// TwinCAT 3 PLC project actuator
// Title: ESO LDC Actuator Library
// Company: ESO
// Author: Dan Popovic
// ProjectVersion: 1.0.0.2
// Description: Local Device Control - LDC Actuator Library based on State Machine
// ProgramVersion: 3.1.0.8
// libraries:
//   Tc2_Standard, * (Beckhoff Automation GmbH)
//   Tc2_System, * (Beckhoff Automation GmbH)
//   Tc2_Utilities, * (Beckhoff Automation GmbH)
//   Tc3_EventLogger, * (Beckhoff Automation GmbH)
//   Tc3_Module, * (Beckhoff Automation GmbH)
//   VisuDialogs, * (System)
// project tree:
//   DUTs/Enumerated/ E_ACTUATOR_RPC_ERROR.TcDUT, E_ACTUATOR_COMMAND.TcDUT, E_ACTUATOR_EVENT.TcDUT, E_ACTUATOR_ERROR.TcDUT, E_ACTUATOR_STATUS.TcDUT, E_ACTUATOR_STATE.TcDUT, E_ACTUATOR_HW_STATUS.TcDUT, E_ACTUATOR_SUBSTATE.TcDUT
//   DUTs/Structures/ T_ACTUATOR_CFG.TcDUT, T_SIM_ACTUATOR_CFG.TcDUT, T_ACTUATOR_CTRL.TcDUT, T_ACTUATOR_INFO.TcDUT, T_ACTUATOR_STAT.TcDUT, T_SIM_ACTUATOR_STAT.TcDUT
//   / GlobalTextList.TcGTLO, PlcTask.TcTTO, Visualization Manager.TcVMO (not stored)
//   POUs/ FB_SIM_ACTUATOR.TcPOU, FB_ACTUATOR.TcPOU, MAIN.TcPOU
//   Version/ Global_Version.TcGVL
//   VISUs/ GUI_Actuator001.TcVIS, GUI_Actuator002.TcVIS, GUI_Actuator003.TcVIS, GUI_Actuator004.TcVIS
//   VISUs/Templates/ GUI_TEMPLATE_ACTUATOR.TcVIS
// real-time tasks:
//   TASK PlcTask: cycle T#1ms, priority 20, ADS port 350
// variable links:
//   actuator/actuator Instance <-> actuator/actuator Instance
//     PlcTask Inputs/MAIN.Actuator001.i_bOn <-> PlcTask Outputs/MAIN.SIM_Actuator001.q_bOn
//     PlcTask Inputs/MAIN.Actuator002.i_bOn <-> PlcTask Outputs/MAIN.SIM_Actuator002.q_bOn
//     PlcTask Inputs/MAIN.Actuator002.i_nCouplerState <-> PlcTask Outputs/MAIN.SIM_Actuator002.q_nCouplerState
//     PlcTask Inputs/MAIN.Actuator003.i_nCouplerState <-> PlcTask Outputs/MAIN.SIM_Actuator003.q_nCouplerState
//     PlcTask Inputs/MAIN.Actuator004.i_nCouplerState <-> PlcTask Outputs/MAIN.SIM_Actuator004.q_nCouplerState
//     PlcTask Inputs/MAIN.SIM_Actuator001.i_bSwitch <-> PlcTask Outputs/MAIN.Actuator001.q_bSwitch
//     PlcTask Inputs/MAIN.SIM_Actuator002.i_bSwitch <-> PlcTask Outputs/MAIN.Actuator002.q_bSwitch
//     PlcTask Inputs/MAIN.SIM_Actuator003.i_bSwitch <-> PlcTask Outputs/MAIN.Actuator003.q_bSwitch
//     PlcTask Outputs/MAIN.Actuator004.q_bSwitch <-> PlcTask Inputs/MAIN.SIM_Actuator004.i_bSwitch
//     PlcTask Outputs/MAIN.SIM_Actuator001.q_nCouplerState <-> PlcTask Inputs/MAIN.Actuator001.i_nCouplerState
//     PlcTask Outputs/MAIN.SIM_Actuator003.q_bOn <-> PlcTask Inputs/MAIN.Actuator003.i_bOn
//     PlcTask Outputs/MAIN.SIM_Actuator004.q_bOn <-> PlcTask Inputs/MAIN.Actuator004.i_bOn

CONFIGURATION actuator
    RESOURCE PLC ON TwinCAT3
        TASK PlcTask(INTERVAL := T#1ms, PRIORITY := 20);
        PROGRAM MAIN WITH PlcTask : MAIN;
    END_RESOURCE
END_CONFIGURATION

// ---- DUTs/Enumerated/E_ACTUATOR_RPC_ERROR.TcDUT
{attribute 'qualified_only'}
{attribute 'strict'}
TYPE E_ACTUATOR_RPC_ERROR :
(
	OK						:= 0,
	NOT_OP					:= -1,			
	NOT_NOTOP_READY			:= -2,			
	NOT_NOTOP				:= -3,			
	SWITCHING_ON			:= -4,			
	SWITCHING_OFF			:= -5,			
	LOCAL					:= -7			
);
END_TYPE

// ---- DUTs/Enumerated/E_ACTUATOR_COMMAND.TcDUT
{attribute 'qualified_only'}
{attribute 'strict'}
TYPE E_ACTUATOR_COMMAND :
(
	NONE	:= 0,
	
	RESET,
	INIT,
	STOP,
	ENABLE,
	DISABLE,
	ON,
	OFF
	
);
END_TYPE

// ---- DUTs/Enumerated/E_ACTUATOR_EVENT.TcDUT
{attribute 'qualified_only'}
{attribute 'strict'}
TYPE E_ACTUATOR_EVENT :
(
	NONE	:= 0,
	
	(* events corresponding to commands *)
	RESET,
	INIT,
	STOP,
	ENABLE,
	DISABLE,
	ON,
	OFF,
	
	(* 
		Events corresponding to internal events 
	*)
	
	INITON,		// Needed for detection of HW failures during initialisation
	INITOFF,
	DISABLEON,
	DISABLEOFF,
	
	(* events mapped to HW signals *)
	ISON,
	ISOFF,

	HWOK,
	ERRHW,
	ERRMAXON,
	ERRTIMEOUT,
	ERRINIT,
	ERRDISABLE
	
);
END_TYPE

// ---- DUTs/Enumerated/E_ACTUATOR_ERROR.TcDUT
{attribute 'qualified_only'}
{attribute 'strict'}
TYPE E_ACTUATOR_ERROR :
(
	OK					:= 0,
	HW_NOTOP,			
	WRONG_CMD,			
	INCONSISTENT,		
	INIT_FAILURE,		
	ENABLE_FAILURE,
	DISABLE_FAILURE,
	ON_FAILURE,
	OFF_FAILURE,
	FAILURE_SIG,
	MAXON,
	STILL_COOLING,
	TIMEOUT,
	// Simulator errors
	NOT_INITIALISED		:= 90,
	ZERO_POINTER		:= 100	
);
END_TYPE

// ---- DUTs/Enumerated/E_ACTUATOR_STATUS.TcDUT
{attribute 'qualified_only'}
{attribute 'strict'}
TYPE E_ACTUATOR_STATUS :
(
	OK	:= 0,
	ERROR
);
END_TYPE

// ---- DUTs/Enumerated/E_ACTUATOR_STATE.TcDUT
{attribute 'qualified_only'}
{attribute 'strict'}
TYPE E_ACTUATOR_STATE :
(
	NONE	:= 0,
	NOTOP,
	OP
);
END_TYPE

// ---- DUTs/Enumerated/E_ACTUATOR_HW_STATUS.TcDUT
{attribute 'qualified_only'}
{attribute 'strict'}
TYPE E_ACTUATOR_HW_STATUS :
(
	UNKNOWN	:= 0,
	ERROR,
	OFF,
	ON
);
END_TYPE

// ---- DUTs/Enumerated/E_ACTUATOR_SUBSTATE.TcDUT
{attribute 'qualified_only'}
{attribute 'strict'}
TYPE E_ACTUATOR_SUBSTATE :
(
	NONE					:= 0,
	
	NOTOP_NOTREADY			:= 100,
	NOTOP_READY_OFF			:= 103,
	NOTOP_READY_ON			:= 104,
	NOTOP_SWITCHING_OFF		:= 109,           
	NOTOP_SWITCHING_ON		:= 110,
	NOTOP_ERROR				:= 199,
	
	OP_OFF					:= 206,            
	OP_SWITCHING_OFF		:= 207,           
	OP_ON					:= 209,
	OP_SWITCHING_ON			:= 210,
	OP_ERROR				:= 299
);
END_TYPE

// ---- DUTs/Structures/T_ACTUATOR_CFG.TcDUT
TYPE T_ACTUATOR_CFG :
STRUCT
	sName:				STRING	:= 'Actuator';// Instance name
	bActiveLowOn:		BOOL 	:= FALSE;	(* If TRUE, On signal is Active Low *)
	bActiveLowSwitch:	BOOL 	:= FALSE;	(* If TRUE, Switch ctrl signal is Active Low *)

	bAutoOp:			BOOL 	:= FALSE;	// If TRUE, go automatically to OPERATIONAL state
	bInitialState:		BOOL 	:= FALSE;	(* default power state is OFF *)
	bInvertAnalog:		BOOL 	:= FALSE;	(* If TRUE, analog feedback is active, if signal < nAnalogThreshold *)
	
	nAnalogThreshold:	DINT 	:= 0;		(* Analog feedback signal threshold [bits].
										   If this signal is used, any value above it will indicate that the power is ON. *)

	nMaxOn:				UDINT 	:= 0;		(* Maximum time for power to be ON [sec] *)
	nSigStablePeriod:   UDINT 	:= 200;		(* signal is stable if it has been constant for so long [msec] *)
	nTimeout:     		UDINT 	:= 5000;	(* timeout for state transitions [msec] *)

	// Logging
	bLogExtTime:		BOOL 	:= FALSE;		// If TRUE, use external time in event logs. Default FALSE.
	bDebug:				BOOL 	:= FALSE;		// If TRUE, show event logs of Debug type. Default FALSE.
	bLog:				BOOL 	:= TRUE;		// If TRUE, log events. Default TRUE.


	
END_STRUCT
END_TYPE

// ---- DUTs/Structures/T_SIM_ACTUATOR_CFG.TcDUT
TYPE T_SIM_ACTUATOR_CFG :
STRUCT
	bActiveLowOn:		BOOL := FALSE;
	bActiveLowSwitch:	BOOL := FALSE;

	nDelay:     		UDINT := 1000;	(* Simulated delay for commands [msec] *)
	
END_STRUCT
END_TYPE

// ---- DUTs/Structures/T_ACTUATOR_CTRL.TcDUT
TYPE T_ACTUATOR_CTRL :
STRUCT
	nCommand:		DINT	:= E_ACTUATOR_COMMAND.NONE;	(* See E_ACTUATOR_COMMAND *)
	bExecute:		BOOL;
	
END_STRUCT
END_TYPE

// ---- DUTs/Structures/T_ACTUATOR_INFO.TcDUT
TYPE T_ACTUATOR_INFO :
STRUCT
(*
Driver Information 

Change Log:
*)
	sDate:			STRING(32)	:= '2018-10-26';
	sDescription:	STRING(80) 	:= 'State Machine based Actuator controller';
	sName:			STRING(64)	:= 'FB_ACTUATOR';
	sPlatform:		STRING(32)	:= 'CoDeSys';
	sSynopsis:		STRING(64)	:= 'State Machine based Actuator controller';
	nVersionMajor:	DINT		:= 1;
	nVersionMinor:	DINT		:= 0;
END_STRUCT
END_TYPE

// ---- DUTs/Structures/T_ACTUATOR_STAT.TcDUT
TYPE T_ACTUATOR_STAT :
STRUCT
	bLocal:			BOOL	:= FALSE;						(* if TRUE, device operated from PLC GUI *)

	nLastCommand:	DINT	:= E_ACTUATOR_COMMAND.NONE;			(* Last command sent to the device *)

	nErrorCode: 	DINT 	:= E_ACTUATOR_ERROR.HW_NOTOP;		(* Error code *)
	nHwStatus: 		DINT	:= E_ACTUATOR_HW_STATUS.UNKNOWN; 		(* Unknown, error, on, of. See E_ACTUATOR_HW_STATUS *)
	nRpcErrorCode: 	DINT	:= E_ACTUATOR_RPC_ERROR.OK;		(* RPC Error code *)
	nStatus: 		DINT	:= E_ACTUATOR_STATUS.ERROR; 			(* Device status *)

	sErrorText: 	STRING 	:= 'OK'; 						(* Error text *)
	sHwStatus: 		STRING 	:= 'UNKNOWN'; 					(* HW Status in textual form: 'UNKNOWN', 'ERROR', 'OPEN' or 'CLOSED' *)
	sLastCommand:	STRING	:= 'NONE';						(* Last command, as string, sent to the device *)
	sLibVersion:	STRING	:= 'UNKNOWN';					(* Library version as string, e.g. '1.2.0.0' *)
	sRPCErrorText: 	STRING 	:= 'OK'; 						(* RPC Error text *)
	sStatus: 		STRING 	:= 'OK'; 						(* Status in textual form, e.g. 'OFF' *)
	
	sState:			STRING	:= 'NOT OP';
	sSubstate:		STRING	:= 'NOT READY';
	
	nState:			E_ACTUATOR_STATE		:= E_ACTUATOR_STATE.NOTOP;
	nSubstate:		E_ACTUATOR_SUBSTATE	:= E_ACTUATOR_SUBSTATE.NOTOP_NOTREADY;
	
	sActionDesc:	STRING	:= '';
	sEventDesc:		STRING	:= '';

	


	nCycleCounter:		UDINT	:= 0;
	nCycleTime:			UDINT	:= 0;						// Cycle time in us (microsec)

	nTimeOn: 			UDINT 	:= 0;						(* Time power has been ON since last ON command [sec] *)
	nTimeOnStart:		UDINT 	:= 0;						(* Absolute start time of last power ON command [sec] *)
	nTimeOnTotal:		UDINT 	:= 0;						(* Total time power has been ON [sec] *)
	nTimeOnTotalStart:	UDINT 	:= 0;						(* Absolute start time of power ON [sec] *)
	nTimeOff: 			UDINT 	:= 0;						(* Time power has been OFF [sec] *)
	nTimeOffStart:		UDINT 	:= 0;						(* Time power has been OFF [sec] *)
	
END_STRUCT
END_TYPE

// ---- DUTs/Structures/T_SIM_ACTUATOR_STAT.TcDUT
TYPE T_SIM_ACTUATOR_STAT :
STRUCT
	bInitialised:	BOOL	:= FALSE;						(* If TRUE, power simulator is initialised *)

	nErrorCode: 	DINT 	:= E_ACTUATOR_ERROR.NOT_INITIALISED;	(* Error code *)
	sErrorText: 	STRING 	:= 'NOT INITIALISED'; 			(* Error text *)
	sStatus: 		STRING 	:= 'ERROR'; 					(* power status in textual form, e.g. 'OFF' *)
END_STRUCT
END_TYPE

// ---- Version/Global_Version.TcGVL
{attribute 'TcGenerated'}
{attribute 'no-analysis'}
{attribute 'linkalways'}
// This function has been automatically generated from the project information.
VAR_GLOBAL CONSTANT
	{attribute 'const_non_replaced'}
	stLibVersion_ESO_LDC_Actuator_Library : ST_LibVersion := (iMajor := 1, iMinor := 0, iBuild := 0, iRevision := 2, nFlags := 0, sVersion := '1.0.0.2');
END_VAR

// ---- POUs/MAIN.TcPOU
PROGRAM MAIN
VAR
	
	{attribute 'OPC.UA.DA':='1'}
	Actuator001:		FB_ACTUATOR;	// Simulated power always
	{attribute 'OPC.UA.DA':='1'}
	Actuator002:		FB_ACTUATOR;	// Simulated power always
	{attribute 'OPC.UA.DA':='1'}
	Actuator003:		FB_ACTUATOR;	// Real power if connected to a PLC
	{attribute 'OPC.UA.DA':='1'}
	Actuator004:		FB_ACTUATOR;	// Real power if connected to a PLC

	{attribute 'OPC.UA.DA':='1'}
	SIM_Actuator001:	FB_SIM_ACTUATOR;
	{attribute 'OPC.UA.DA':='1'}
	SIM_Actuator002:	FB_SIM_ACTUATOR;
	{attribute 'OPC.UA.DA':='1'}
	SIM_Actuator003:	FB_SIM_ACTUATOR;
	{attribute 'OPC.UA.DA':='1'}
	SIM_Actuator004:	FB_SIM_ACTUATOR;
	
END_VAR

// Actuator001 configuration:
// - Go to  OPERATIONAL on PLC reboot
// - Initial state is OFF
Actuator001(in_sName:='Actuator001', in_bAutoOp:=TRUE,in_bInitialState:=FALSE);

// Actuator002 configuration:
// - Go to  OPERATIONAL on PLC reboot
// - Initial state is ON
Actuator002(in_sName:='Actuator002', in_bAutoOp:=TRUE,in_bInitialState:=TRUE);

// Actuator003 configuration:
// - Remain in NOTOP on PLC reboot
// - Initial state is OFF
Actuator003(in_sName:='Actuator003', in_bAutoOp:=FALSE,in_bInitialState:=FALSE);

// Actuator004 configuration:
// - Go to  OPERATIONAL on PLC reboot
// - Initial state is ON
Actuator004(in_sName:='Actuator004', in_bAutoOp:=TRUE,in_bInitialState:=TRUE);


// Actuator001 Simulator
SIM_Actuator001(ptrDev:=ADR(Actuator001));
// Actuator002 Simulator
SIM_Actuator002(ptrDev:=ADR(Actuator002));
// Actuator003 Simulator
SIM_Actuator003(ptrDev:=ADR(Actuator003));
// Actuator004 Simulator
SIM_Actuator004(ptrDev:=ADR(Actuator004));

END_PROGRAM

// ---- POUs/FB_ACTUATOR.TcPOU
FUNCTION_BLOCK FB_ACTUATOR
VAR_INPUT
	{attribute 'OPC.UA.DA' := '0'}
	in_sName:				STRING	:= 'Actuator';	// Default device name

	{attribute 'OPC.UA.DA' := '0'}
	in_bActiveLowOn:		BOOL	:= FALSE;	// If TRUE, On signal is Active Low. Default FALSE.
	{attribute 'OPC.UA.DA' := '0'}
	in_bActiveLowSwitch:	BOOL 	:= FALSE;	// If TRUE, Switch ctrl signal is Active Low. Default FALSE.

	{attribute 'OPC.UA.DA' := '0'}
	in_bAutoOp:				BOOL 	:= FALSE;	// If TRUE, go automatically to OPERATIONAL state. Default FALSE.
	{attribute 'OPC.UA.DA' := '0'}
	in_bInitialState:		BOOL 	:= FALSE;	// Default power state is OFF (FALSE).
	{attribute 'OPC.UA.DA' := '0'}
	in_bInvertAnalog:		BOOL 	:= FALSE;	// If TRUE, analog feedback is active if signal < nAnalogThreshold. Default FALSE.
	
	{attribute 'OPC.UA.DA' := '0'}
	in_nAnalogThreshold:	DINT 	:= 0;		// Analog feedback signal threshold [bits]. Used if <>0. Default 0, i.e. not used.
												// If this signal is used, any value above it will indicate that the power is ON.
	{attribute 'OPC.UA.DA' := '0'}
	in_nMaxOn:				UDINT 	:= 0;		// Maximum time for power to be ON [sec]. Default 0, no limit.
	{attribute 'OPC.UA.DA' := '0'}
	in_nSigStablePeriod:	UDINT 	:= 200;		// Signal is stable if it has been constant for so long [msec]. Default 200 ms.
	{attribute 'OPC.UA.DA' := '0'}
	in_nTimeout:     		UDINT 	:= 5000;	// Timeout for state transitions [msec]. Default 5000 ms (5 sec).
END_VAR
VAR_OUTPUT
END_VAR
VAR
	{attribute 'OPC.UA.DA' := '1'}
	cfg:		T_ACTUATOR_CFG;	
	{attribute 'OPC.UA.DA' := '1'}
	ctrl:		T_ACTUATOR_CTRL;	
	{attribute 'OPC.UA.DA' := '1'}
	{attribute 'OPC.UA.DA.Access' := '1'}
	info:		T_ACTUATOR_INFO;				// ReadOnly
	{attribute 'OPC.UA.DA' := '1'}
	{attribute 'OPC.UA.DA.Access' := '1'}
	stat:		T_ACTUATOR_STAT;				// ReadOnly

	{attribute 'OPC.UA.DA' := '0'}
	nEvent:		      	DINT := E_ACTUATOR_EVENT.NONE;
	{attribute 'OPC.UA.DA' := '0'}
	nInternalEvent:		DINT := E_ACTUATOR_EVENT.NONE;
	
	// Operational Events
	{attribute 'OPC.UA.DA' := '0'}
	fbEventStart:	FB_TcMessage;
	{attribute 'OPC.UA.DA' := '0'}
	fbEventEnd:		FB_TcMessage;
	{attribute 'OPC.UA.DA' := '0'}
	fbEventError:	FB_TcMessage;
	{attribute 'OPC.UA.DA' := '0'}
	fbEventDebug:	FB_TcMessage;
	{attribute 'OPC.UA.DA' := '0'}
	fbEventGeneral:	FB_TcMessage;
	
	
	(***** Local variables *****)
	{attribute 'OPC.UA.DA' := '0'}
	bOn:		BOOL;						// Feedback - combination of digital and analog
	{attribute 'OPC.UA.DA' := '0'}
	toutCmd:	TON;
	{attribute 'OPC.UA.DA' := '0'}
	trg:		R_TRIG;
	{attribute 'OPC.UA.DA' := '0'}
	timer:		TON;						// Timer for measuring duration of events
	


	///// Physical signals - to be mapped!!! /////

	// Outputs
	{attribute 'OPC.UA.DA' := '0'}
	q_bSwitch 		AT %Q*: 		BOOL;	// power control digital output

	// Inputs	
	{attribute 'OPC.UA.DA' := '0'}
	i_nCouplerState	AT %I*: 		UINT;	// Link it to Coupler->InfoData->State
	{attribute 'OPC.UA.DA' := '0'}
	i_bOn 			AT %I*: 		BOOL;	// Digital feedback signal
	{attribute 'OPC.UA.DA' := '0'}
	i_nOn			AT %I*: 		INT;	// Analog feedback signal

	// Flag if the device is ready to receive commands.
	// It takes about 3.5 sec for the system to go OPERATIONAL.
	{attribute 'OPC.UA.DA' := '0'}
	bDeviceReady:		BOOL 	:= FALSE;
END_VAR

IF NOT bDeviceReady THEN
	// Set device Configuration
	M_Configure();
	RETURN;
END_IF

// Increment counter.
// This will be seen as 'alive' flag.
stat.nCycleCounter	:= stat.nCycleCounter + 1;



(* === Check for commands and internal events to be processed === *)
CheckForEvents();

(* === Process events according to the State Machine === *)
ProcessEvents();

METHOD ActionErrExecute
VAR
END_VAR
SetAction('ActionErrExecute');

IF nEvent = E_ACTUATOR_EVENT.ERRTIMEOUT THEN
	stat.nErrorCode		:= E_ACTUATOR_ERROR.ON_FAILURE;
	stat.sErrorText		:= 'ERROR: Timeout';	
END_IF
END_METHOD

METHOD ActionInitAbort
VAR_INPUT
END_VAR
SetAction('ActionInitAbort');

(* reply Error *)
stat.nErrorCode		:= E_ACTUATOR_ERROR.INIT_FAILURE;
stat.sErrorText		:= 'ERROR: INIT command aborted due to STOP or RESET.';

(* Reset the timer for the command *)
toutCmd(IN:=FALSE);
END_METHOD

METHOD ActionInitExecute
VAR_INPUT
END_VAR
VAR
	nCurrentTime:	UDINT;
END_VAR
SetAction('ActionInitExecute');

// Log event
M_LogEventStart('INIT');

(* reply OK *)
stat.nErrorCode		:= E_ACTUATOR_ERROR.OK;
stat.sErrorText		:= 'OK';

(* Reset the timer action *)
toutCmd(IN:=FALSE);

nCurrentTime			:= GetTimeInSec();
stat.nTimeOffStart		:= nCurrentTime;
UpdateTimes(bOnState:=FALSE, bRestart:=FALSE, bReset:=FALSE);

// Do not touch the outputs.
// Just change the state depending on the status
IF bOn THEN
	SetState(E_ACTUATOR_STATE.NOTOP, E_ACTUATOR_SUBSTATE.NOTOP_READY_ON);
ELSE
	SetState(E_ACTUATOR_STATE.NOTOP, E_ACTUATOR_SUBSTATE.NOTOP_READY_OFF);
END_IF
END_METHOD

METHOD ActionInitReject
VAR_INPUT
END_VAR
SetAction('ActionInitReject');

(* Reject an INIT command since another one is in progress. *)
(* do not reset the timer ... *)
END_METHOD

METHOD ActionMaxOnFailure
VAR_INPUT
END_VAR
(* code to initiate the switching OFF of the power *)
SetAction('ActionMaxOnFailure');

// Log event
M_LogEventError('Actuator maximum ON time exceeded.. Switched to OFF.');

(* Set the error *)
SetStatus(E_ACTUATOR_ERROR.MAXON,'ERROR: Actuator maximum ON time exceeded.');

UpdateTimes(bOnState:=FALSE, bRestart:=TRUE, bReset:=FALSE);


(* Switch power OFF *)
q_bSwitch	:= GetLogicalState(FALSE, cfg.bActiveLowSwitch);

(* 
	Reset signal trigger and its timer. 
	Next transition activity, e.g. ActivitySwitchingOff, will complete when the signal has been OFF 
	for longer than cfg.nSigStablePeriod [ms].
*)
trg(CLK:=FALSE);
timer(IN:=FALSE);	// Timer for stable signal lasting cfg.nSigStablePeriod

(* Restart the command timer *)
toutCmd(IN:=FALSE);
toutCmd(IN:=TRUE,PT:=UDINT_TO_TIME(cfg.nTimeout));
END_METHOD

METHOD ActionOffExecute
VAR_INPUT
END_VAR
(* code to initiate the switching OFF of the power *)
SetAction('ActionOffExecute');

// Log event
M_LogEventStart('OFF');

(* Clear the error *)
SetStatus(E_ACTUATOR_ERROR.OK,'OK');

UpdateTimes(bOnState:=FALSE, bRestart:=TRUE, bReset:=FALSE);


(* Actuator power OFF *)
q_bSwitch	:= GetLogicalState(FALSE, cfg.bActiveLowSwitch);

(* 
	Reset signal trigger and its timer. 
	Next transition activity, e.g. ActivitySwitchingOff, will complete when the signal has been OFF 
	for longer than cfg.nSigStablePeriod [ms].
*)
trg(CLK:=FALSE);
timer(IN:=FALSE);	// Timer for stable signal lasting cfg.nSigStablePeriod

(* Restart the command timer *)
toutCmd(IN:=FALSE);
toutCmd(IN:=TRUE,PT:=UDINT_TO_TIME(cfg.nTimeout));
END_METHOD

METHOD ActionOnExecute
VAR_INPUT
END_VAR
(* Code to initiate turning the power ON *)

SetAction('ActionOnExecute');

// Log event
M_LogEventStart('ON');

(* Clear the error *)
SetStatus(E_ACTUATOR_ERROR.OK,'OK');

(* Turn the control signal ON  *)
q_bSwitch	:= GetLogicalState(TRUE, cfg.bActiveLowSwitch);


(* 
	Reset signal trigger and its timer. 
	Next transition activity, e.g. ActivitySwitchingOn, will complete when the signal has been ON 
	for longer than cfg.nSigStablePeriod [ms].
*)
trg(CLK:=FALSE);
timer(IN:=FALSE);	// Timer for stable signal lasting cfg.nSigStablePeriod

(* Start the timer for command timeout of cfg.nTimeout *)
toutCmd(IN:=FALSE);	
toutCmd(IN:=TRUE,PT:=UDINT_TO_TIME(cfg.nTimeout));
END_METHOD

METHOD ActionResetExecute
VAR_INPUT
END_VAR
SetAction('ActionResetExecute');

// Log event
M_LogEventStart('RESET');

(* reply Error *)
SetStatus(nErrorCode:=E_ACTUATOR_ERROR.OK, sErrorText:='OK');

// Go to the default state on PLC re-boot
q_bSwitch	:= GetLogicalState(cfg.bInitialState, cfg.bActiveLowSwitch);

// Reset ON/OFF times
UpdateTimes(bOnState:=bOn,bRestart:=FALSE,bReset:=TRUE);	

(* Reset the timer for the command *)
toutCmd(IN:=FALSE);

// In ActionOnExecute() and ActionOffExecute(), we are waiting for trg() to go from FALSE to TRUE.
// Trigger it with FALSE.
trg(CLK:=FALSE);

IF cfg.bInitialState = TRUE THEN
	ActionOnExecute();
	SetState(E_ACTUATOR_STATE.NOTOP, E_ACTUATOR_SUBSTATE.NOTOP_SWITCHING_ON);
ELSE
	ActionOffExecute();
	SetState(E_ACTUATOR_STATE.NOTOP, E_ACTUATOR_SUBSTATE.NOTOP_SWITCHING_OFF);
END_IF
END_METHOD

METHOD ActionUnexpExecute
VAR
END_VAR
SetAction('ActionUnexpExecute');

IF nEvent = E_ACTUATOR_EVENT.ISON THEN
	IF	stat.nLastCommand = E_ACTUATOR_COMMAND.ON 	AND
		stat.nSubstate = E_ACTUATOR_SUBSTATE.OP_OFF 	AND
		stat.nErrorCode = E_ACTUATOR_ERROR.TIMEOUT		THEN
		M_LogEventGeneral('Recovered after timeout. Actuator is ON');
	END_IF
ELSIF nEvent = E_ACTUATOR_EVENT.ISOFF THEN
	IF	stat.nLastCommand = E_ACTUATOR_COMMAND.OFF 	AND
		stat.nSubstate = E_ACTUATOR_SUBSTATE.OP_ON 	AND
		stat.nErrorCode = E_ACTUATOR_ERROR.TIMEOUT		THEN
		M_LogEventGeneral('Recovered after timeout. Actuator is OFF');
	END_IF
ELSIF nEvent = E_ACTUATOR_EVENT.ON THEN
	stat.nErrorCode		:= E_ACTUATOR_ERROR.STILL_COOLING;
	stat.sErrorText		:= 'ERROR: ON command not allowed while cooling.';	
	stat.sStatus		:= 'ERROR';	
	stat.nStatus		:= E_ACTUATOR_STATUS.ERROR;
END_IF
END_METHOD

METHOD ActivityOff
VAR_INPUT
END_VAR
SetAction('ActivityOff');

// Update the OFF time
UpdateTimes(bOnState:=FALSE, bRestart:=FALSE, bReset:=FALSE);
END_METHOD

METHOD ActivityOn
VAR_INPUT
END_VAR
SetAction('ActivityOn');

// Update the ON time
UpdateTimes(bOnState:=TRUE, bRestart:=FALSE, bReset:=FALSE);
END_METHOD

METHOD ActivitySwitchingOff
VAR_INPUT
END_VAR
(* 
	This activity monitors the OFF power task and 
	triggers the ISOFF event at completion. 
*)
SetAction('ActivitySwitchingOff');


(* 
	The signal has to be OFF for longer than cfg.nSigStablePeriod [msec].
	The timer will start when bOn=FALSE trigger is detected.
*)
(* Execute trigger - note the 'NOT bOn' detectiong the transition from ON to OFF *)
trg(CLK := NOT bOn);

IF trg.Q THEN
	(* Restart the signal duration timer *)
	timer(IN:=FALSE);
	timer(IN:=TRUE,PT:=UDINT_TO_TIME(cfg.nSigStablePeriod));
END_IF

(* Execute signal duration timer *)
timer();

IF	timer.Q OR 
	((NOT bOn) AND cfg.nSigStablePeriod = 0) THEN
	timer(IN:=FALSE);	// Reset the signal duration timer
	toutCmd(IN:=FALSE);	// Reset the command timeout timer

	(* Update time ON/OFF *)
	UpdateTimes(bOnState:=TRUE, bRestart:=FALSE, bReset:=FALSE);

	(* 
		Normally, we would go to state E_SWITCH_SUBSTATE.OP_COOLING. 
		However, if the cooldown time is zero, i.e. no cooldown, we go directly to state E_ACTUATOR_SUBSTATE.OP_OFF.
	*)
	nInternalEvent 		:= E_ACTUATOR_EVENT.ISOFF;
	
	// Log event
	M_LogEventEnd('OFF');

//	stat.nErrorCode		:= E_ACTUATOR_ERROR.OK;
//	stat.sErrorText		:= 'OK';	

	RETURN;
END_IF

(* 
	if the timeout is detected before reaching the position, 
	then trigger the internal error event 
*)
toutCmd();
IF toutCmd.Q THEN
	toutCmd(IN:=FALSE);	(* Reset Timer *)
	timer(IN:=FALSE);	(* Reset the signal duration timer *)
	
	nInternalEvent  := E_ACTUATOR_EVENT.ERRTIMEOUT;
	SetStatus(E_ACTUATOR_ERROR.TIMEOUT, 'ERROR: Switching OFF timed out.');

	// Log event
	M_LogEventError('OFF command timed out');
END_IF
END_METHOD

METHOD ActivitySwitchingOn
VAR_INPUT
END_VAR
(* 
	This activity to monitor the ON power task and 
	trigger the ISON event at completion. 
*)
SetAction('ActivitySwitchingOn');

(* 
	The signal has to be ON for longer than cfg.nSigStablePeriod [msec].
	The timer will start when bOn trigger is detected.
*)
(* Execute trigger *)
trg(CLK:=bOn);

IF trg.Q THEN
	(* Restart the signal duration timer *)
	timer(IN:=FALSE);
	timer(IN:=TRUE,PT:=UDINT_TO_TIME(cfg.nSigStablePeriod));
END_IF

(* Execute signal duration timer *)
timer();

IF	timer.Q OR 
	(bOn AND cfg.nSigStablePeriod = 0) THEN
	timer(IN:=FALSE);	// Reset the signal duration timer
	toutCmd(IN:=FALSE);	// Reset the command timeout timer

	(* Update time ON/OFF *)
	IF stat.nTimeOn > 0 THEN
		// power was already ON, restart the ON time.
		UpdateTimes(bOnState:=TRUE, bRestart:=TRUE, bReset:=FALSE);
	ELSE
		// power was OFF, don't restart the ON time.
		UpdateTimes(bOnState:=TRUE, bRestart:=FALSE, bReset:=FALSE);
	END_IF

	(* 
		Normally, we would go to state E_ACTUATOR_SUBSTATE.OP_WARMING. 
		However, if the warmup time is zero, i.e. no warmup, we go directly to state E_ACTUATOR_SUBSTATE.OP_ON.
	*)
	nInternalEvent 		:= E_ACTUATOR_EVENT.ISON;	
	
	// Log event
	M_LogEventEnd('ON');

	stat.nErrorCode		:= E_ACTUATOR_ERROR.OK;
	stat.sErrorText		:= 'OK';	

	RETURN;
END_IF

(* 
	if the timeout is detected before reaching the position, 
	then trigger the internal error event 
*)
toutCmd();
IF toutCmd.Q THEN
	toutCmd(IN:=FALSE);	(* Reset Timer *)
	timer(IN:=FALSE);	(* Reset the signal duration timer *)
	
	nInternalEvent  := E_ACTUATOR_EVENT.ERRTIMEOUT;
	SetStatus(E_ACTUATOR_ERROR.TIMEOUT, 'ERROR: Switching ON timed out.');

	// Log event
	M_LogEventError('ON command timed out');

END_IF
END_METHOD

METHOD CheckForEvents
VAR_INPUT
END_VAR

(* 
	Start assuming the HW is OK. 
	This is needed to recover from the situation where 
	the HW was failing and now it is working.
*)
nEvent := E_ACTUATOR_EVENT.HWOK;


(*
	Read all inputs, i.e. get status of INPUT signals based on ActiveLow configuration 
*)


(* The power ON feedback can be analog and/or digital. *)
IF 	(GetLogicalState(i_bOn, cfg.bActiveLowOn)) OR
	(cfg.nAnalogThreshold <> 0 AND (i_nOn > cfg.nAnalogThreshold) AND NOT cfg.bInvertAnalog) OR
	(cfg.nAnalogThreshold <> 0 AND (i_nOn < cfg.nAnalogThreshold) AND     cfg.bInvertAnalog)	THEN
	bOn	:= TRUE;
ELSE
	bOn	:= FALSE;
END_IF


UpdateTimes(bOnState:=bOn,bRestart:=FALSE, bReset:=FALSE);	// Update the Time


(* HW Status in textual form: 'ERROR', 'ON' or 'OFF' *)
IF 		bOn   = TRUE  THEN
	stat.nHwStatus	:= E_ACTUATOR_HW_STATUS.ON;
	stat.sHwStatus	:= 'ON';
ELSIF 	bOn   = FALSE  THEN
	stat.nHwStatus	:= E_ACTUATOR_HW_STATUS.OFF;
	stat.sHwStatus	:= 'OFF';
END_IF

(* 
	Check for events in the following order: 
   	1) HW failure: without HW avilability there is no point to do anything
	2) Internal events: to allow completing the initiated commands before 
                        starting processing new commands. 
   	3) Commands: to react to external commands. Commands should be executed 
                 before processing HW signals to allow to start a recovery action.
   	4) HW signals:  such as power is ON/OFF.
*)

IF i_nCouplerState <> 8 THEN	
	(* Check if the HW is NOT OK *)
	(*
	If the hardware status is NOT OK, we cannot trust the readings.
	Variable i_nCouplerState has to be mapped to a State of a terminal, e.g. EK1100.
	The value should be 8.
 	*)
	SetEvent(E_ACTUATOR_EVENT.ERRHW);
	SetStatus(E_ACTUATOR_ERROR.HW_NOTOP, 'ERROR: HW not in OPERATIONAL state');
	RETURN;

ELSIF nInternalEvent <> E_ACTUATOR_EVENT.NONE THEN
	(* Handle internal events *)
	SetEvent(nInternalEvent);
	nInternalEvent := E_ACTUATOR_EVENT.NONE;
ELSIF ctrl.bExecute = TRUE  THEN
	(* Handle commands *)
	ctrl.bExecute		:= FALSE;			(* Clear the Execute bit *)
	SetLastCommand(ctrl.nCommand);			(* Save the last command *)
	SetEvent(ctrl.nCommand);
	ctrl.nCommand 		:= E_ACTUATOR_COMMAND.NONE;	(* Clear the Command *)
ELSE
	(* Handle HW problems and unexpected bahaviour *)
	
	IF stat.nSubstate = E_ACTUATOR_SUBSTATE.NOTOP_READY_OFF OR 
	   stat.nSubstate = E_ACTUATOR_SUBSTATE.NOTOP_READY_ON OR 
	   stat.nSubstate = E_ACTUATOR_SUBSTATE.OP_OFF OR 
	   stat.nSubstate = E_ACTUATOR_SUBSTATE.OP_ON OR 
	   stat.nSubstate = E_ACTUATOR_SUBSTATE.OP_ERROR THEN
	   
		(* Set events for ON and OFF *)		
		IF	bOn   = TRUE  THEN
			SetEvent(E_ACTUATOR_EVENT.ISON);
		ELSIF	bOn   = FALSE THEN
			SetEvent(E_ACTUATOR_EVENT.ISOFF);
		END_IF	
	END_IF	
(*
	IF stat.nSubstate = E_ACTUATOR_SUBSTATE.OP_SWITCHING_ON THEN
		(* Set events for ON  *)		
		IF	bOn   = TRUE  THEN
			SetEvent(E_ACTUATOR_EVENT.ISON);
		END_IF	
	END_IF	
	*)
END_IF
END_METHOD

METHOD GetLogicalState : BOOL
(*
	This method returns the state of the variable based on its 
	activeLow configuration.
	Syntax:
		bState	:= GetLogicalState (<var value>,  <activeLow cfg>);
		
	Example 1:
		var = TRUE;
		activeLow = FALSE;
		bState	:= GetLogicalState (TRUE,  FALSE); = TRUE

	Example 2:
		var = TRUE;
		activeLow = TRUE;
		bState	:= GetLogicalState (TRUE,  TRUE); = FALSE
*)
VAR_INPUT
	state:		BOOL;
	activeLow:	BOOL;
END_VAR
IF activeLow THEN
	GetLogicalState := NOT state;
ELSE
	GetLogicalState := state;
END_IF
END_METHOD

METHOD GetTimeInSec : UDINT
(*
	This method returns absolute time in seconds.
*)
(* System time is given in 100ns. Divide by 10000000 to get in seconds. *)
GetTimeInSec := ULINT_TO_UDINT(Tc2_System.F_GetSystemTime() / 10000000);
END_METHOD

METHOD M_Configure : BOOL
VAR_INPUT
END_VAR
VAR
     fbGetCurTaskIdx:	GETCURTASKINDEX;
END_VAR
// If device is ready, there is nothing to configure.
IF bDeviceReady THEN
	RETURN;
END_IF

// If first cycle, copy configuration AND RETURN in order for the system to read all inputs before doing any work
IF stat.nCycleCounter = 0 THEN
	
	// Copy input parameters into configuration
	cfg.sName				:=	in_sName;			

	cfg.bActiveLowOn		:= in_bActiveLowOn;
	cfg.bActiveLowSwitch	:= in_bActiveLowSwitch;
	cfg.bAutoOp				:= in_bAutoOp;
	cfg.bInitialState		:= in_bInitialState;
	cfg.bInvertAnalog		:= in_bInvertAnalog;
	cfg.nAnalogThreshold	:= in_nAnalogThreshold;
	cfg.nMaxOn				:= in_nMaxOn;
	cfg.nSigStablePeriod	:= in_nSigStablePeriod;
	cfg.nTimeout			:= in_nTimeout;
	
	// Get the version number 
	stat.sLibVersion	:= stLibVersion_ESO_LDC_Actuator_Library.sVersion;

	// Get cycle time in microsec.
	// CycleTime in _TaskInfo is given in 100 ns. 1 us = 1000 ns
	fbGetCurTaskIdx();
	stat.nCycleTime	:=  (TwinCAT_SystemInfoVarList._TaskInfo[fbGetCurTaskIdx.index].CycleTime)/10;
	
	// Increment counter.
	stat.nCycleCounter	:= stat.nCycleCounter + 1;
	RETURN;
ELSIF (stat.nCycleCounter * stat.nCycleTime) < 5000000 THEN
	// EtherCAT is normally ready after 3.5 sec.
	// We give it 5 sec to consider it to be ready.
	// Increment counter.
	stat.nCycleCounter	:= stat.nCycleCounter + 1;
	RETURN;
END_IF


// Create Event instances
fbEventStart.CreateEx	(TC_EVENTS.ActuatorOpsEventClass.ActionStart,0);
fbEventEnd.CreateEx		(TC_EVENTS.ActuatorOpsEventClass.ActionEnd,0);
fbEventError.CreateEx	(TC_EVENTS.ActuatorOpsEventClass.Error,0);
fbEventDebug.CreateEx	(TC_EVENTS.ActuatorOpsEventClass.Debug,0);
fbEventGeneral.CreateEx	(TC_EVENTS.ActuatorOpsEventClass.General,0);

// The device is ready now.
bDeviceReady := TRUE;


// Clear errors
stat.nErrorCode		:= E_ACTUATOR_ERROR.OK;
stat.sErrorText		:= 'OK';	


//
// Set next state based on cfg.bAutoOp
//

// Go to the default state on PLC re-boot.
// Default state is set in cfg.bInitialState.
q_bSwitch	:= GetLogicalState(cfg.bInitialState, cfg.bActiveLowSwitch);

// In ActionOnExecute() and ActionOffExecute(), we are waiting for trg() to go from FALSE to TRUE.
// Trigger it with FALSE.
trg(CLK:=FALSE);

// Go directly to the target state.
IF NOT cfg.bAutoOp THEN
	// Go automatically to NOTOP ON or OFF
	IF cfg.bInitialState = TRUE THEN
		ActionOnExecute();
		SetState(E_ACTUATOR_STATE.NOTOP, E_ACTUATOR_SUBSTATE.NOTOP_SWITCHING_ON);
	ELSE
		ActionOffExecute();
		SetState(E_ACTUATOR_STATE.NOTOP, E_ACTUATOR_SUBSTATE.NOTOP_SWITCHING_OFF);
	END_IF
ELSE
	// Go automatically to OPERATIONAL
	// If initial state is ON, go to E_ACTUATOR_SUBSTATE.OP_SWITCHING_ON.
	// Otherwise, go to E_ACTUATOR_SUBSTATE.OP_SWITCHING_OFF.
	IF cfg.bInitialState = TRUE THEN
		ActionOnExecute();
		SetState(E_ACTUATOR_STATE.OP, E_ACTUATOR_SUBSTATE.OP_SWITCHING_ON);
	ELSE
		ActionOffExecute();
		SetState(E_ACTUATOR_STATE.OP, E_ACTUATOR_SUBSTATE.OP_SWITCHING_OFF);
	END_IF
END_IF
END_METHOD

METHOD M_GetRpcErrorText : STRING
VAR_INPUT
	ErrorCode:	INT;
END_VAR
VAR
	str:	STRING;
END_VAR
CASE ErrorCode OF
	E_ACTUATOR_RPC_ERROR.OK:					str	:= 'OK';
	E_ACTUATOR_RPC_ERROR.NOT_OP:				str	:= 'Cannot control device. Not in OP state.';
	E_ACTUATOR_RPC_ERROR.NOT_NOTOP_READY:		str	:= 'Call failed. Not in NOTOP_READY.';
	E_ACTUATOR_RPC_ERROR.NOT_NOTOP:				str	:= 'Call failed. Not in NOTOP.';
	E_ACTUATOR_RPC_ERROR.SWITCHING_ON:			str	:= 'Device OFF failed. Still switching ON.';
	E_ACTUATOR_RPC_ERROR.SWITCHING_OFF:			str	:= 'Device ON failed. Still switching OFF.';
	E_ACTUATOR_RPC_ERROR.LOCAL:					str	:= 'RPC calls not allowed in Local mode.';
ELSE
	str	:= 'Unregistered RPC error.';
END_CASE

M_GetRpcErrorText	:= str;
END_METHOD

METHOD M_LogEventDebug : BOOL
VAR_INPUT
	sText:	STRING	:= '';
END_VAR
// Log Debug events only if both logging and debugging is enabled
IF  cfg.bLog AND cfg.bDebug THEN
	fbEventDebug.ipArguments.Clear().AddString(sText);
	fbEventDebug.Send(0);
END_IF
END_METHOD

METHOD M_LogEventEnd : BOOL
VAR_INPUT
	sText:	STRING	:= '';
END_VAR
// Log only if logging is enabled
IF  NOT cfg.bLog THEN
	RETURN;
END_IF

fbEventEnd.ipArguments.Clear().AddString(sText);
fbEventEnd.Send(0);
END_METHOD

METHOD M_LogEventError : BOOL
VAR_INPUT
	sText:	STRING	:= '';
END_VAR
// Log only if logging is enabled
IF  NOT cfg.bLog THEN
	RETURN;
END_IF

fbEventError.ipArguments.Clear().AddString(sText);
fbEventError.Send(0);
END_METHOD

METHOD M_LogEventGeneral : BOOL
VAR_INPUT
	sText:	STRING	:= '';
END_VAR
// Log only if logging is enabled
IF  NOT cfg.bLog THEN
	RETURN;
END_IF

fbEventGeneral.ipArguments.Clear().AddString(sText);
fbEventGeneral.Send(0);
END_METHOD

METHOD M_LogEventStart : BOOL
VAR_INPUT
	sText:	STRING	:= '';
END_VAR
// Log only if logging is enabled
IF  NOT cfg.bLog THEN
	RETURN;
END_IF

fbEventStart.ipArguments.Clear().AddString(sText);
fbEventStart.Send(0);
END_METHOD

METHOD M_SetRpcStatus : INT
VAR_INPUT
	nErrorCode:	E_ACTUATOR_RPC_ERROR;
END_VAR
stat.nRpcErrorCode	:= nErrorCode;
stat.sRpcErrorText	:= M_GetRpcErrorText(nErrorCode);

M_SetRpcStatus		:= nErrorCode;
END_METHOD

METHOD ProcessEvents
VAR_INPUT
END_VAR

VAR
END_VAR
(* 
	Before processing the event, execute the Do-Activity tasks. 
	Note that, in case of orthogonal regions, more than one Do-Activity 
	could run in the same PLC cycle.
	Note: Most of these activities have timeouts since they take time.
*)

IF 	stat.nSubstate = E_ACTUATOR_SUBSTATE.NOTOP_SWITCHING_ON  OR  
	stat.nSubstate = E_ACTUATOR_SUBSTATE.OP_SWITCHING_ON 		THEN
	ActivitySwitchingOn();
END_IF

IF stat.nSubstate = E_ACTUATOR_SUBSTATE.OP_ON THEN
	ActivityOn();	// Just update times
END_IF

IF 	stat.nSubstate = E_ACTUATOR_SUBSTATE.NOTOP_SWITCHING_OFF  OR  
	stat.nSubstate = E_ACTUATOR_SUBSTATE.OP_SWITCHING_OFF 		THEN
	ActivitySwitchingOff();
END_IF

IF stat.nSubstate = E_ACTUATOR_SUBSTATE.OP_OFF THEN
	ActivityOff();	// Just update times
END_IF


(* 
	Evaluate state machine transitions.
*)

CASE stat.nState OF

//***********************************
// NOTOP
//***********************************
E_ACTUATOR_STATE.NOTOP:

	(* Transitions from NOTOP substates *)
	CASE stat.nSubstate OF
	
	E_ACTUATOR_SUBSTATE.NOTOP_NOTREADY:
		// This state should not exist.
		// Go to ON or OFF immediately.		
		// ActionResetExecute() will do it for us.
		ActionResetExecute();
		RETURN;
		
	E_ACTUATOR_SUBSTATE.NOTOP_SWITCHING_OFF:		// TODO	
		IF nEvent = E_ACTUATOR_EVENT.STOP THEN
			ActionInitAbort();
			SetState(E_ACTUATOR_STATE.NOTOP, E_ACTUATOR_SUBSTATE.NOTOP_NOTREADY);
			RETURN;
		ELSIF nEvent = E_ACTUATOR_EVENT.ERRINIT THEN
			M_LogEventError('INIT failed');
			SetState(E_ACTUATOR_STATE.NOTOP, E_ACTUATOR_SUBSTATE.NOTOP_NOTREADY);
			RETURN;
		ELSIF nEvent = E_ACTUATOR_EVENT.INITOFF THEN
			SetState(E_ACTUATOR_STATE.NOTOP, E_ACTUATOR_SUBSTATE.NOTOP_READY_OFF);
			RETURN;
		ELSIF nEvent = E_ACTUATOR_EVENT.ISOFF THEN
			SetState(E_ACTUATOR_STATE.NOTOP, E_ACTUATOR_SUBSTATE.NOTOP_READY_OFF);
			RETURN;
		END_IF
		
	E_ACTUATOR_SUBSTATE.NOTOP_SWITCHING_ON:		// TODO	
		IF nEvent = E_ACTUATOR_EVENT.STOP THEN
			ActionInitAbort();
			SetState(E_ACTUATOR_STATE.NOTOP, E_ACTUATOR_SUBSTATE.NOTOP_NOTREADY);
			RETURN;
		ELSIF nEvent = E_ACTUATOR_EVENT.ERRINIT THEN
			M_LogEventError('INIT failed');
			SetState(E_ACTUATOR_STATE.NOTOP, E_ACTUATOR_SUBSTATE.NOTOP_NOTREADY);
			RETURN;
		ELSIF nEvent = E_ACTUATOR_EVENT.INITOFF THEN
			SetState(E_ACTUATOR_STATE.NOTOP, E_ACTUATOR_SUBSTATE.NOTOP_READY_OFF);
			RETURN;
		ELSIF nEvent = E_ACTUATOR_EVENT.ISON THEN
			SetState(E_ACTUATOR_STATE.NOTOP, E_ACTUATOR_SUBSTATE.NOTOP_READY_ON);
			RETURN;
		ELSIF nEvent = E_ACTUATOR_EVENT.INITON THEN
			SetState(E_ACTUATOR_STATE.NOTOP, E_ACTUATOR_SUBSTATE.NOTOP_READY_ON);
			RETURN;
		END_IF
		
	E_ACTUATOR_SUBSTATE.NOTOP_READY_OFF:			
		IF nEvent = E_ACTUATOR_EVENT.ISON THEN
			ActionUnexpExecute();
			SetState(E_ACTUATOR_STATE.NOTOP, E_ACTUATOR_SUBSTATE.NOTOP_READY_ON);
			RETURN;
		ELSIF nEvent = E_ACTUATOR_EVENT.ENABLE THEN
			SetAction('ActionEnableExecute');
			M_LogEventGeneral('Enabled');
			SetState(E_ACTUATOR_STATE.OP, E_ACTUATOR_SUBSTATE.OP_OFF);
			RETURN;
		END_IF

	E_ACTUATOR_SUBSTATE.NOTOP_READY_ON:			
		IF nEvent = E_ACTUATOR_EVENT.ISOFF THEN
			ActionUnexpExecute();
			SetState(E_ACTUATOR_STATE.NOTOP, E_ACTUATOR_SUBSTATE.NOTOP_READY_OFF);
			RETURN;
		ELSIF nEvent = E_ACTUATOR_EVENT.ENABLE THEN
			SetAction('ActionEnableExecute');
			M_LogEventGeneral('Enabled');
			SetState(E_ACTUATOR_STATE.OP, E_ACTUATOR_SUBSTATE.OP_ON);
			RETURN;
		END_IF

	E_ACTUATOR_SUBSTATE.NOTOP_ERROR:			
		IF nEvent = E_ACTUATOR_EVENT.HWOK THEN
			M_LogEventGeneral('Recovered from ERROR state. HW is OK');
			SetState(E_ACTUATOR_STATE.NOTOP, E_ACTUATOR_SUBSTATE.NOTOP_NOTREADY);
			RETURN;
		END_IF
		
	END_CASE

	(* Transitions from NOTOP state *)
	IF nEvent = E_ACTUATOR_EVENT.ERRHW THEN
		// Log the error only once
		IF stat.nSubstate <> E_ACTUATOR_SUBSTATE.NOTOP_ERROR THEN
			M_LogEventError('HW not in OPERATIONAL state');
		END_IF
		SetStatus(E_ACTUATOR_ERROR.HW_NOTOP, 'ERROR: HW not in OPERATIONAL state');
		SetState(E_ACTUATOR_STATE.NOTOP, E_ACTUATOR_SUBSTATE.NOTOP_ERROR);
		RETURN;
	END_IF
	
//***********************************
// OPERATIONAL
//***********************************
E_ACTUATOR_STATE.OP:

	(* Transitions from OP substates *)
	CASE stat.nSubstate OF
	E_ACTUATOR_SUBSTATE.OP_OFF:			
		IF nEvent = E_ACTUATOR_EVENT.ON THEN
			ActionOnExecute();
			SetState(E_ACTUATOR_STATE.OP, E_ACTUATOR_SUBSTATE.OP_SWITCHING_ON);
			RETURN;
		ELSIF nEvent = E_ACTUATOR_EVENT.OFF THEN
			// Nothing to do. Just clear previous error, if any.
			SetStatus(E_ACTUATOR_ERROR.OK, 'OK');
			M_LogEventGeneral('Command OFF ignored. Already OFF');
			RETURN;
		ELSIF nEvent = E_ACTUATOR_EVENT.ISON THEN
			ActionUnexpExecute();
			SetState(E_ACTUATOR_STATE.OP, E_ACTUATOR_SUBSTATE.OP_ON);
			RETURN;
		ELSIF nEvent = E_ACTUATOR_EVENT.DISABLE THEN
			M_LogEventGeneral('Disabled');
			SetState(E_ACTUATOR_STATE.NOTOP, E_ACTUATOR_SUBSTATE.NOTOP_READY_OFF);
			RETURN;		
		END_IF

	E_ACTUATOR_SUBSTATE.OP_SWITCHING_ON:			
		IF nEvent = E_ACTUATOR_EVENT.ISON THEN
			SetState(E_ACTUATOR_STATE.OP, E_ACTUATOR_SUBSTATE.OP_ON);
			RETURN;
		ELSIF nEvent = E_ACTUATOR_EVENT.ON THEN
			// Clear previous error, if any.
			SetStatus(E_ACTUATOR_ERROR.OK, 'OK');
			// Log event
			M_LogEventGeneral('New ON command. Restarted Time ON counter.');
			// Restart the TimeON
			UpdateTimes(bOnState:=TRUE,bRestart:=TRUE, bReset:=FALSE);
			RETURN;
		ELSIF nEvent = E_ACTUATOR_EVENT.ERRTIMEOUT THEN
			SetState(E_ACTUATOR_STATE.OP, E_ACTUATOR_SUBSTATE.OP_ERROR);
			RETURN;
		END_IF
		
	E_ACTUATOR_SUBSTATE.OP_ON:			
		IF nEvent = E_ACTUATOR_EVENT.OFF THEN
			ActionOffExecute();
			SetState(E_ACTUATOR_STATE.OP, E_ACTUATOR_SUBSTATE.OP_SWITCHING_OFF);
			RETURN;
		ELSIF nEvent = E_ACTUATOR_EVENT.ON THEN
			// Clear previous error, if any.
			SetStatus(E_ACTUATOR_ERROR.OK, 'OK');
			// Log event
			M_LogEventGeneral('New ON command. Restarted Time ON counter.');
			// Restart the TimeON
			UpdateTimes(bOnState:=TRUE,bRestart:=TRUE, bReset:=FALSE);
			RETURN;
		ELSIF nEvent = E_ACTUATOR_EVENT.ISOFF THEN
			ActionUnexpExecute();
			SetState(E_ACTUATOR_STATE.OP, E_ACTUATOR_SUBSTATE.OP_OFF);
			RETURN;
		ELSIF nEvent = E_ACTUATOR_EVENT.DISABLE THEN
			M_LogEventGeneral('Disabled');
			SetState(E_ACTUATOR_STATE.NOTOP, E_ACTUATOR_SUBSTATE.NOTOP_READY_ON);
			RETURN;	
		ELSIF nEvent = E_ACTUATOR_EVENT.ERRMAXON THEN
			ActionMaxOnFailure();
			SetState(E_ACTUATOR_STATE.OP, E_ACTUATOR_SUBSTATE.OP_SWITCHING_OFF);
			RETURN;				
		END_IF
		
	E_ACTUATOR_SUBSTATE.OP_SWITCHING_OFF:			
		IF nEvent = E_ACTUATOR_EVENT.ISOFF THEN
			SetState(E_ACTUATOR_STATE.OP, E_ACTUATOR_SUBSTATE.OP_OFF);
			RETURN;
		ELSIF nEvent = E_ACTUATOR_EVENT.ERRTIMEOUT THEN
			SetState(E_ACTUATOR_STATE.OP, E_ACTUATOR_SUBSTATE.OP_ERROR);
			RETURN;
		END_IF
		
	E_ACTUATOR_SUBSTATE.OP_ERROR:			
		IF nEvent = E_ACTUATOR_EVENT.OFF THEN
			ActionOffExecute();
			SetState(E_ACTUATOR_STATE.OP, E_ACTUATOR_SUBSTATE.OP_SWITCHING_OFF);
			RETURN;
		ELSIF nEvent = E_ACTUATOR_EVENT.ON THEN
			ActionOnExecute();
			SetState(E_ACTUATOR_STATE.OP, E_ACTUATOR_SUBSTATE.OP_SWITCHING_ON);
			RETURN;			
		ELSIF nEvent = E_ACTUATOR_EVENT.ISON THEN
			IF stat.nErrorCode <> E_ACTUATOR_ERROR.HW_NOTOP THEN
				SetStatus(E_ACTUATOR_ERROR.OK, 'OK');	// Clear error
			ELSE
				M_LogEventGeneral('Recovered from ERROR state. Actuator is ON');
			END_IF
			SetState(E_ACTUATOR_STATE.OP, E_ACTUATOR_SUBSTATE.OP_ON);
			RETURN;			
		ELSIF nEvent = E_ACTUATOR_EVENT.ISOFF THEN
			IF stat.nErrorCode <> E_ACTUATOR_ERROR.HW_NOTOP THEN
				SetStatus(E_ACTUATOR_ERROR.OK, 'OK');	// Clear error
			ELSE
				M_LogEventGeneral('Recovered from ERROR state. Actuator is OFF');
			END_IF
			SetState(E_ACTUATOR_STATE.OP, E_ACTUATOR_SUBSTATE.OP_OFF);
			RETURN;	
		ELSIF nEvent = E_ACTUATOR_EVENT.DISABLE THEN
			IF bOn THEN
				SetState(E_ACTUATOR_STATE.NOTOP, E_ACTUATOR_SUBSTATE.NOTOP_READY_ON);
			ELSE
				SetState(E_ACTUATOR_STATE.NOTOP, E_ACTUATOR_SUBSTATE.NOTOP_READY_OFF);
			END_IF
			RETURN;			
		END_IF

	END_CASE
	
	(* Transitions from OP state *)
	IF nEvent = E_ACTUATOR_EVENT.ERRHW THEN
		IF stat.nSubstate <> E_ACTUATOR_SUBSTATE.OP_ERROR THEN
			// Log the error only once
			M_LogEventError('HW not in OPERATIONAL state');
		END_IF
		SetStatus(E_ACTUATOR_ERROR.HW_NOTOP, 'ERROR: HW not in OPERATIONAL state');
		SetState(E_ACTUATOR_STATE.OP, E_ACTUATOR_SUBSTATE.OP_ERROR);

		RETURN;
	END_IF
	
END_CASE

(* 
	"Global" internal transitions valid in any state should go here.
	They do not change the active state configuration. 
	They are evaluated after all the others transitions have been 
	considered.
*) 
IF nEvent = E_ACTUATOR_EVENT.RESET THEN
	ActionResetExecute();
	RETURN;
ELSIF nEvent = E_ACTUATOR_EVENT.STOP THEN
	RETURN;
END_IF
END_METHOD

{attribute 'TcRpcEnable':='1'}
METHOD RPC_Disable : INT
VAR_INPUT
END_VAR
// RPC calls are not allowed in Local mode.
IF stat.bLocal THEN
	RPC_Disable	:= M_SetRpcStatus(E_ACTUATOR_RPC_ERROR.LOCAL);
	RETURN;
END_IF

// Disable command is accepted only if device is in OP state.
IF stat.nState <> E_ACTUATOR_STATE.OP THEN
	RPC_Disable	:= M_SetRpcStatus(E_ACTUATOR_RPC_ERROR.NOT_OP);
	RETURN;
ELSE
	// Clear RPC Call status
	stat.sRPCErrorText	:= 'OK';
	
	// Set disable command
	ctrl.nCommand := E_ACTUATOR_COMMAND.DISABLE;
	ctrl.bExecute := TRUE;
	
	// Call was successful
	RPC_Disable	:= M_SetRpcStatus(E_ACTUATOR_RPC_ERROR.OK);
END_IF
END_METHOD

{attribute 'TcRpcEnable':='1'}
METHOD RPC_Enable : INT
VAR_INPUT
END_VAR
// RPC calls are not allowed in Local mode.
IF stat.bLocal THEN
	RPC_Enable	:= M_SetRpcStatus(E_ACTUATOR_RPC_ERROR.LOCAL);
	RETURN;
END_IF

// Enable command is accepted only if device is in NOTOP_READY.
IF	stat.nState = E_ACTUATOR_STATE.NOTOP					AND  
	stat.nSubstate <> E_ACTUATOR_SUBSTATE.NOTOP_READY_OFF	AND  
	stat.nSubstate <> E_ACTUATOR_SUBSTATE.NOTOP_READY_ON		THEN
	RPC_Enable	:= M_SetRpcStatus(E_ACTUATOR_RPC_ERROR.NOT_NOTOP_READY);
	RETURN;
ELSE
	// Clear RPC Call status
	stat.sRPCErrorText	:= 'OK';
	
	// Set enable command
	ctrl.nCommand := E_ACTUATOR_COMMAND.ENABLE;
	ctrl.bExecute := TRUE;
	
	// Call was successful
	RPC_Enable	:= M_SetRpcStatus(E_ACTUATOR_RPC_ERROR.OK);
END_IF
END_METHOD

{attribute 'TcRpcEnable':='1'}
METHOD RPC_Init : INT
VAR_INPUT
END_VAR
// RPC calls are not allowed in Local mode.
IF stat.bLocal THEN
	RPC_Init	:= M_SetRpcStatus(E_ACTUATOR_RPC_ERROR.LOCAL);
	RETURN;
END_IF

// Init command is accepted only in NOTOP.
IF	stat.nState <> E_ACTUATOR_STATE.NOTOP	THEN
	RPC_Init	:= M_SetRpcStatus(E_ACTUATOR_RPC_ERROR.NOT_NOTOP);
	RETURN;
ELSE
	// Clear RPC Call status
	stat.sRPCErrorText	:= 'OK';
	
	// Set INIT command
	ctrl.nCommand := E_ACTUATOR_COMMAND.INIT;
	ctrl.bExecute := TRUE;
	
	// Call was successful
	RPC_Init	:= M_SetRpcStatus(E_ACTUATOR_RPC_ERROR.OK);
END_IF
END_METHOD

{attribute 'TcRpcEnable':='1'}
METHOD RPC_Off : INT
VAR_INPUT
END_VAR
// RPC calls are not allowed in Local mode.
IF stat.bLocal THEN
	RPC_Off	:= M_SetRpcStatus(E_ACTUATOR_RPC_ERROR.LOCAL);
	RETURN;
END_IF

// OFF command is accepted only in OP state.
IF	stat.nState <> E_ACTUATOR_STATE.OP	THEN
	RPC_Off	:= M_SetRpcStatus(E_ACTUATOR_RPC_ERROR.NOT_OP);
	RETURN;
ELSIF stat.nSubstate = E_ACTUATOR_SUBSTATE.OP_SWITCHING_ON THEN
	// power should not be commanded to go OFF if being switched ON.
	RPC_Off	:= M_SetRpcStatus(E_ACTUATOR_RPC_ERROR.SWITCHING_ON);
	RETURN;
ELSE
	// Clear RPC Call status
	stat.sRPCErrorText	:= 'OK';
	
	// Set OFF command
	ctrl.nCommand := E_ACTUATOR_COMMAND.OFF;
	ctrl.bExecute := TRUE;
	
	// Call was successful
	RPC_Off	:= M_SetRpcStatus(E_ACTUATOR_RPC_ERROR.OK);
END_IF
END_METHOD

{attribute 'TcRpcEnable':='1'}
METHOD RPC_On : INT
VAR_INPUT
END_VAR
// RPC calls are not allowed in Local mode.
IF stat.bLocal THEN
	RPC_On	:= M_SetRpcStatus(E_ACTUATOR_RPC_ERROR.LOCAL);
	RETURN;
END_IF

// ON command is accepted only in OP state and NOT COOLING.
IF	stat.nState <> E_ACTUATOR_STATE.OP	THEN
	RPC_On	:= M_SetRpcStatus(E_ACTUATOR_RPC_ERROR.NOT_OP);
	RETURN;
ELSIF stat.nSubstate = E_ACTUATOR_SUBSTATE.OP_SWITCHING_OFF THEN
	// power should not be commanded to go ON if being switched OFF.
	RPC_On	:= M_SetRpcStatus(E_ACTUATOR_RPC_ERROR.SWITCHING_OFF);
	RETURN;
ELSE
	// Clear RPC Call status
	stat.sRPCErrorText	:= 'OK';
	
	// Set ON command
	ctrl.nCommand 		:= E_ACTUATOR_COMMAND.ON;
	ctrl.bExecute 		:= TRUE;
	
	// Call was successful
	RPC_On	:= M_SetRpcStatus(E_ACTUATOR_RPC_ERROR.OK);
END_IF
END_METHOD

{attribute 'TcRpcEnable':='1'}
METHOD RPC_Reset : INT
VAR_INPUT
END_VAR
// RPC calls are not allowed in Local mode.
IF stat.bLocal THEN
	RPC_Reset	:= M_SetRpcStatus(E_ACTUATOR_RPC_ERROR.LOCAL);
	RETURN;
END_IF

// Clear RPC Call status
stat.sRPCErrorText	:= 'OK';

ctrl.nCommand := E_ACTUATOR_COMMAND.RESET;
ctrl.bExecute := TRUE;

// Call was successful
RPC_Reset	:= M_SetRpcStatus(E_ACTUATOR_RPC_ERROR.OK);
END_METHOD

{attribute 'TcRpcEnable':='1'}
METHOD RPC_Stop : INT
VAR_INPUT
END_VAR
// RPC calls are not allowed in Local mode.
IF stat.bLocal THEN
	RPC_Stop	:= M_SetRpcStatus(E_ACTUATOR_RPC_ERROR.LOCAL);
	RETURN;
END_IF

// Clear RPC Call status
stat.sRPCErrorText	:= 'OK';

ctrl.nCommand := E_ACTUATOR_COMMAND.STOP;
ctrl.bExecute := TRUE;

// Call was successful
RPC_Stop	:= M_SetRpcStatus(E_ACTUATOR_RPC_ERROR.OK);
END_METHOD

METHOD SetAction
VAR_INPUT
	actionName:		STRING;
END_VAR


stat.sActionDesc := actionName;
END_METHOD

METHOD SetEvent
VAR_INPUT
	nEventId:			DINT;
END_VAR

nEvent := nEventId;

CASE nEventId OF
	E_ACTUATOR_EVENT.NONE:
		stat.sEventDesc := '';
		RETURN;
		
	E_ACTUATOR_EVENT.RESET:
		stat.sEventDesc := 'CMD RESET';
		RETURN;
	
	E_ACTUATOR_EVENT.INIT:
		stat.sEventDesc := 'CMD INIT';
		RETURN;

	E_ACTUATOR_EVENT.STOP:
		stat.sEventDesc := 'CMD STOP';
		RETURN;

	E_ACTUATOR_EVENT.ENABLE:
		stat.sEventDesc := 'CMD ENABLE';
		RETURN;

	E_ACTUATOR_EVENT.DISABLE:
		stat.sEventDesc := 'CMD DISABLE';
		RETURN;

	E_ACTUATOR_EVENT.ON:
		stat.sEventDesc := 'CMD ON';
		RETURN;

	E_ACTUATOR_EVENT.OFF:
		stat.sEventDesc := 'CMD OFF';
		RETURN;
	
	(* events corresponding to internal events *)
	E_ACTUATOR_EVENT.INITOFF:
		stat.sEventDesc := 'INT INITOFF';
		RETURN;

	E_ACTUATOR_EVENT.INITON:
		stat.sEventDesc := 'INT INITON';
		RETURN;

	E_ACTUATOR_EVENT.DISABLEOFF:
		stat.sEventDesc := 'INT DISABLEOFF';
		RETURN;
	
	E_ACTUATOR_EVENT.DISABLEON:
		stat.sEventDesc := 'INT DISABLEON';
		RETURN;
	
	(* evetnts mapped to HW signals *)
	E_ACTUATOR_EVENT.ISON:
		stat.sEventDesc := 'SIG ISON';
		RETURN;

	E_ACTUATOR_EVENT.ISOFF:
		stat.sEventDesc := 'SIG ISOFF';
		RETURN;

	E_ACTUATOR_EVENT.HWOK:
		stat.sEventDesc := 'SIG HWOK';
		RETURN;

	E_ACTUATOR_EVENT.ERRHW:
		stat.sEventDesc := 'INT ERRHW';
		RETURN;

	E_ACTUATOR_EVENT.ERRMAXON:	
		stat.sEventDesc := 'INT ERRMAXON';
		RETURN;

	E_ACTUATOR_EVENT.ERRTIMEOUT:	
		stat.sEventDesc := 'INT ERRTIMEOUT';
		RETURN;

	E_ACTUATOR_EVENT.ERRINIT:
		stat.sEventDesc := 'INT ERRINIT';
		RETURN;

	E_ACTUATOR_EVENT.ERRDISABLE:
		stat.sEventDesc := 'INT ERRDISABLE';
		RETURN;
	
END_CASE 

(* INTERNAL ERROR *)
stat.sEventDesc := 'UNKNOWN EVENT';
END_METHOD

METHOD SetLastCommand
VAR_INPUT
	cmd:	DINT;
END_VAR
stat.nLastCommand	:= cmd;

CASE cmd OF
	E_ACTUATOR_COMMAND.RESET:
		stat.sLastCommand	:= 'RESET';
	E_ACTUATOR_COMMAND.INIT:
		stat.sLastCommand	:= 'INIT';
	E_ACTUATOR_COMMAND.STOP:
		stat.sLastCommand	:= 'STOP';
	E_ACTUATOR_COMMAND.ENABLE:
		stat.sLastCommand	:= 'ENABLE';
	E_ACTUATOR_COMMAND.DISABLE:
		stat.sLastCommand	:= 'DISABLE';
	E_ACTUATOR_COMMAND.ON:
		stat.sLastCommand	:= 'ON';
	E_ACTUATOR_COMMAND.OFF:
		stat.sLastCommand	:= 'OFF';
ELSE
		stat.sLastCommand	:= 'NONE';
END_CASE;
END_METHOD

METHOD SetState : BOOL
VAR_INPUT
	nState:			E_ACTUATOR_STATE;
	nSubstate:		E_ACTUATOR_SUBSTATE;
END_VAR
(* 
	Update State Machine active state configuration.

	ToDo: support initial pseudo state/substate.
*)

IF nState <> E_ACTUATOR_STATE.NONE THEN
	stat.nState	:= nState;
END_IF
IF nSubstate <> E_ACTUATOR_SUBSTATE.NONE THEN
	stat.nSubstate	:= nSubstate;
END_IF

(* Update active state configuration description *)

IF nState = E_ACTUATOR_STATE.NOTOP THEN
	stat.sState	:= 'NOT OP';
ELSIF nState = E_ACTUATOR_STATE.OP THEN
	stat.sState	:= 'OPERATIONAL';
END_IF

IF nSubstate = E_ACTUATOR_SUBSTATE.NOTOP_NOTREADY THEN
	stat.sSubstate	:= 'NOT READY';
ELSIF nSubstate = E_ACTUATOR_SUBSTATE.NOTOP_SWITCHING_OFF THEN
	stat.sSubstate	:= 'SWITCHING OFF';
ELSIF nSubstate = E_ACTUATOR_SUBSTATE.NOTOP_SWITCHING_ON THEN
	stat.sSubstate	:= 'SWITCHING ON';
ELSIF nSubstate = E_ACTUATOR_SUBSTATE.NOTOP_READY_OFF THEN
	stat.sSubstate	:= 'READY OFF';
ELSIF nSubstate = E_ACTUATOR_SUBSTATE.NOTOP_READY_ON THEN
	stat.sSubstate	:= 'READY ON';
ELSIF nSubstate = E_ACTUATOR_SUBSTATE.NOTOP_ERROR THEN
	stat.sSubstate	:= 'ERROR';
ELSIF nSubstate = E_ACTUATOR_SUBSTATE.OP_OFF THEN
	stat.sSubstate	:= 'OFF';
ELSIF nSubstate = E_ACTUATOR_SUBSTATE.OP_ON THEN
	stat.sSubstate	:= 'ON';
ELSIF nSubstate = E_ACTUATOR_SUBSTATE.OP_SWITCHING_OFF THEN
	stat.sSubstate	:= 'SWITCHING OFF';
ELSIF nSubstate = E_ACTUATOR_SUBSTATE.OP_SWITCHING_ON THEN
	stat.sSubstate	:= 'SWITCHING ON';
ELSIF nSubstate = E_ACTUATOR_SUBSTATE.OP_ERROR THEN
	stat.sSubstate	:= 'ERROR';
ELSE
	stat.sSubstate	:= '';
END_IF


SetState	:= TRUE;
END_METHOD

METHOD SetStatus
VAR_INPUT
	nErrorCode:	DINT;
	sErrorText:	STRING;
END_VAR
stat.nErrorCode 	:= nErrorCode;
stat.sErrorText 	:= sErrorText;

IF nErrorCode <> E_ACTUATOR_ERROR.OK THEN
	stat.sStatus	:= 'ERROR';
	stat.nStatus	:= E_ACTUATOR_STATUS.ERROR;
ELSE
	stat.sStatus	:= 'OK';
	stat.nStatus	:= E_ACTUATOR_STATUS.OK;
END_IF
END_METHOD

METHOD UpdateTimes
VAR_INPUT
	bOnState:	BOOL;	// State of ON status signal
	bRestart:	BOOL := FALSE;	// If TRUE, restart ON time after new command
	bReset:		BOOL := FALSE;	// If TRUE, reset ON /OFF times
END_VAR
VAR
	nCurrentTime:	UDINT;
END_VAR
nCurrentTime	:= GetTimeInSec();

IF bReset OR stat.nSubstate = E_ACTUATOR_SUBSTATE.NOTOP_NOTREADY THEN
	stat.nTimeOnStart		:= nCurrentTime;
	stat.nTimeOnTotalStart	:= nCurrentTime;
	stat.nTimeOffStart		:= nCurrentTime;
	stat.nTimeOnTotal		:= 0;
	stat.nTimeOn			:= 0;
	stat.nTimeOff			:= 0;
	RETURN;
END_IF


IF bOnState THEN
	// power state is ON.
	// In order to avoid OFF time jumps, reset OFF start time.
	stat.nTimeOffStart	:= nCurrentTime;
	
	// Check if the power has already been ON.
	IF	stat.nSubstate = E_ACTUATOR_SUBSTATE.OP_ON THEN
		// power has already been ON
		stat.nTimeOnTotal	:= nCurrentTime - stat.nTimeOnTotalStart;

		IF bRestart THEN
			stat.nTimeOnStart	:= nCurrentTime;
			stat.nTimeOn		:= 0;
		ELSE
			stat.nTimeOn		:= nCurrentTime - stat.nTimeOnStart;
		END_IF
	ELSE
		// power has been OFF
		stat.nTimeOnStart		:= nCurrentTime;
		stat.nTimeOnTotalStart	:= nCurrentTime;
		stat.nTimeOnTotal		:= 0;
		stat.nTimeOn			:= 0;
		stat.nTimeOff			:= 0;
	END_IF

	// Check if the power has been ON for too long, i.e. cfg.nMaxOn exceeded.
	IF stat.nTimeOn > cfg.nMaxOn AND cfg.nMaxOn > 0 THEN
		nInternalEvent  := E_ACTUATOR_EVENT.ERRMAXON;
		RETURN;
	END_IF

ELSE
	// power state is OFF.
	// In order to avoid OFF time jumps, reset OFF start time.
	stat.nTimeOnStart	:= nCurrentTime;
	
	// Check if the power has already been OFF.
	IF 	stat.nSubstate = E_ACTUATOR_SUBSTATE.OP_OFF THEN
		// power has already been OFF
		stat.nTimeOff	:= nCurrentTime - stat.nTimeOffStart;
	ELSE
		IF bRestart THEN
			stat.nTimeOffStart	:= nCurrentTime;
			stat.nTimeOff		:= 0;
		ELSE
			stat.nTimeOff		:= nCurrentTime - stat.nTimeOffStart;
		END_IF
	END_IF
END_IF
END_METHOD

END_FUNCTION_BLOCK

// ---- POUs/FB_SIM_ACTUATOR.TcPOU
FUNCTION_BLOCK FB_SIM_ACTUATOR
VAR_INPUT
	ptrDev:		POINTER TO FB_ACTUATOR;
END_VAR
VAR_OUTPUT
END_VAR
VAR
	{attribute 'OPC.UA.DA':='0'}
	ptrCfg:		POINTER TO T_ACTUATOR_CFG;
	{attribute 'OPC.UA.DA':='0'}
	ptrStat:	POINTER TO T_ACTUATOR_STAT;

	{attribute 'OPC.UA.DA':='1'}
	cfg:			T_SIM_ACTUATOR_CFG;		(* ActiveLow configuration for each signal *)
	{attribute 'OPC.UA.DA':='1'}
	stat:			T_SIM_ACTUATOR_STAT;	(* Simulator status parameters *)
	
	{attribute 'OPC.UA.DA':='0'}
	bSwitch:		BOOL := FALSE;
	{attribute 'OPC.UA.DA':='0'}
	bSwitchLast:	BOOL := FALSE;
	
	{attribute 'OPC.UA.DA':='0'}
	bOn:			BOOL := TRUE;
	{attribute 'OPC.UA.DA':='0'}
	nCouplerState:	UINT := 8;       // normal coupler state
	
    (* Inputs *)
	{attribute 'OPC.UA.DA':='0'}
	i_bSwitch 		AT %I*: 	BOOL;

	(* Outputs *)	
	{attribute 'OPC.UA.DA':='0'}
	q_bOn 		AT %Q*: 		BOOL;
	{attribute 'OPC.UA.DA':='0'}
	q_nCouplerState AT %Q*:		UINT := 8;
	
	{attribute 'OPC.UA.DA':='0'}
	timer:			TON;
	
	{attribute 'OPC.UA.DA':='0'}
	trigger:		R_TRIG;	// To capture device INIT
	
END_VAR

IF NOT stat.bInitialised THEN
	ptrCfg	:= ADR(ptrDev^.cfg);
	ptrStat	:= ADR(ptrDev^.stat);

	// Check for NULL pointers in input parameters
	IF ptrCfg = 0  OR  ptrStat = 0 THEN
		stat.nErrorCode	:= E_ACTUATOR_ERROR.ZERO_POINTER;
		stat.sErrorText	:= 'ERROR: Input parameter is a NULL pointer';
		stat.sStatus	:= 'ERROR';
		RETURN;
	END_IF

	RPC_ResetConfig();	// Copy configuration from device
	
	timer(IN:=FALSE);
	timer(IN:=TRUE,PT:=UDINT_TO_TIME(100));	// Update almost immediately

	stat.nErrorCode	:= E_ACTUATOR_ERROR.OK;
	stat.sErrorText	:= 'OK';
	stat.sStatus	:= 'OK';
	
	stat.bInitialised	:= TRUE;
	RETURN;
END_IF

// There are two triggers: 
// 	Detect device INIT
// 	Activation of switch

// Check for INIT trigger
//trigger(CLK:=(ptrStat^.sActionDesc = 'ActionInitExecute'));
trigger(CLK:=(	ptrStat^.nSubstate=E_ACTUATOR_SUBSTATE.NOTOP_SWITCHING_ON OR 
				ptrStat^.nSubstate=E_ACTUATOR_SUBSTATE.NOTOP_SWITCHING_OFF));

// Get the state of control command
bSwitch := GetLogicalState(i_bSwitch, cfg.bActiveLowSwitch);

IF trigger.Q THEN
	RPC_ResetConfig();	// Copy configuration from device
ELSIF bSwitch <> bSwitchLast THEN
	// Switch value has changed. 
	bSwitchLast	:= bSwitch;
	// Delayed response
	timer(IN:=FALSE);
	timer(IN:=TRUE,PT:=UDINT_TO_TIME(cfg.nDelay));
END_IF


// Execute the timer
timer();

// Set new outputs once the timer has expired
IF timer.Q THEN
	timer(IN:=FALSE);	// Reset timer
	// Set output, i.e. feedback
	bOn	:= GetLogicalState(bSwitch,	cfg.bActiveLowOn);
END_IF


(* Assign outputs *)
q_bOn 			:= bOn;
q_nCouplerState := nCouplerState;

METHOD GetLogicalState : BOOL
(*
	This method returns the state of the variable based on its 
	activeLow configuration.
	Syntax:
		bState	:= GetLogicalState (<var value>,  <activeLow cfg>);
		
	Example 1:
		var = TRUE;
		activeLow = FALSE;
		bState	:= GetLogicalState (TRUE,  FALSE); = TRUE

	Example 2:
		var = TRUE;
		activeLow = TRUE;
		bState	:= GetLogicalState (TRUE,  TRUE); = FALSE
*)
VAR_INPUT
	state:		BOOL;
	activeLow:	BOOL;
END_VAR
IF activeLow THEN
	GetLogicalState := NOT state;
ELSE
	GetLogicalState := state;
END_IF
END_METHOD

{attribute 'TcRpcEnable':='1'}
METHOD RPC_ResetConfig : BOOL
VAR_INPUT
END_VAR
cfg.bActiveLowOn		:= ptrCfg^.bActiveLowOn;
cfg.bActiveLowSwitch	:= ptrCfg^.bActiveLowSwitch;
// Response delay = 1/2 of real switch timeout - the stable signal period
cfg.nDelay				:= ptrCfg^.nTimeout / 2 - ptrCfg^.nSigStablePeriod;	
IF cfg.nDelay < 0 THEN
	cfg.nDelay	:= 0;
END_IF
nCouplerState			:= 8;

// Get the Switch value
bSwitch := GetLogicalState(i_bSwitch, cfg.bActiveLowSwitch);

bOn	:= GetLogicalState(bSwitch,	cfg.bActiveLowOn);	// Set Switch state

RPC_ResetConfig	:= TRUE;
END_METHOD

{attribute 'TcRpcEnable':='1'}
METHOD RPC_SetActiveLow_On : BOOL
VAR_INPUT
	bValue:	BOOL;
END_VAR
cfg.bActiveLowOn	:= bValue;

RPC_SetActiveLow_On	:= TRUE;
END_METHOD

{attribute 'TcRpcEnable':='1'}
METHOD RPC_SetActiveLow_Switch : BOOL
VAR_INPUT
	bValue:	BOOL;
END_VAR
cfg.bActiveLowSwitch	:= bValue;

RPC_SetActiveLow_Switch	:= TRUE;
END_METHOD

{attribute 'TcRpcEnable':='1'}
METHOD RPC_SetCouplerState : BOOL
VAR_INPUT
	bValue:	UINT;
END_VAR
nCouplerState	:= bValue;

RPC_SetCouplerState	:= TRUE;
END_METHOD

{attribute 'TcRpcEnable':='1'}
METHOD RPC_SetDelay : BOOL
VAR_INPUT
	nDelay:	UDINT;	// Response delay [msec]
END_VAR
cfg.nDelay	:= nDelay;

RPC_SetDelay	:= TRUE;
END_METHOD

END_FUNCTION_BLOCK

// ---- GlobalTextList.TcGTLO
TEXTLIST GlobalTextList
  46 = '%.0f'
  23 = '%d'
  62 = '%d sec '
  13 = '%s'
  451 = "'Actuator.library version'"
  386 = "'IODev.library version'"
  857 = "'Switch.library version'"
  77 = 'A period of time [ms] that the feedback signal has to have constant value before taking its status.'
  78 = 'A period of time [ms] that the feedback signal has to have constant value before taking its status.\nMinimum 10 ms.'
  26 = 'Action'
  8 = 'ACTIVATE'
  36 = 'Active Low'
  67 = 'Actual power intensity [%] (0..100)'
  70 = 'Analog feedback signal threshold [bit].\nIf used, the threshold should be > 0.\n'
  71 = 'AnalogThreshold [bit]'
  39 = 'Checkbox'
  15 = 'CLOSE'
  35 = 'Configuration'
  56 = 'Control'
  58 = 'Cooldown'
  53 = 'Cooldown time [sec]  (>=0). \nZero means no cooldown.\n'
  50 = 'Cooldown [sec]'
  9 = 'DEACTIVATE'
  7 = 'DISABLE'
  6 = 'ENABLE'
  74 = 'Error Code'
  535 = 'Error code. Zero means no error.'
  19 = 'Error Description'
  27 = 'Event'
  40 = 'Fault'
  345 = 'Feedback Timeout [ms]'
  73 = 'Feedback Timeout [sec]'
  63 = 'Full range of A/D converter controlling the intensity [bit]  (>=0). \n'
  55 = 'Full range of A/D converter controlling the intensity [bit].\nExamples:\n12 bit A/D = 4095\n15 bit A/D = 32767 \n16 bit A/D = 65535\n'
  52 = 'Full range [bit]'
  61 = 'GREEN means state is active'
  69 = 'GUI disabled !!!\nActivate "Local Control".'
  22 = 'HW'
  28 = 'HW Status'
  113 = 'If checked, logging is active.'
  819 = 'If checked, switch is active on PLC reboot and after RESET.'
  627 = 'If checked, switch is automatically turned ON on PLC reboot and after RESET.'
  234 = 'If checked, switch is automatically turned ON on PLC reboot or after RESET.'
  397 = 'If checked, switch is ON on PLC reboot and after RESET.'
  500 = 'If the logic is inverted, the actuator is considered to be ON, if the reading is below the threshold.'
  107 = 'If the logic is inverted, the lamp is considered to be ON, if the reading is below the threshold.'
  44 = 'If the logic is inverted, the power is considered to be ON, if the reading is below the threshold.'
  89 = 'If the logic is inverted, the switch is considered to be ON, if the reading is below the threshold.'
  37 = 'Ignore'
  38 = 'Ignore Fault'
  4 = 'INIT'
  765 = 'Initial State'
  64 = 'Intensity [%]'
  43 = 'Inver Analog Logic'
  45 = 'Invert Analog Logic'
  16 = 'ISOPEN'
  66 = 'Lamp has to be initialised before it can be used.\n\nRED = not initialised\nGREEN = initialised\n'
  65 = 'Local Control'
  127 = 'Log'
  51 = 'Max ON [sec]'
  851 = 'Maximum allowed time for actuator to be ON [sec]  (>=0). \nZero means no limit.\n'
  54 = 'Maximum allowed time for lamp to be ON [sec]  (>=0). \nZero means no limit.\n'
  300 = 'Maximum allowed time for switch to be ON [sec]  (>=0). \nZero means no limit.\n'
  17 = 'not used'
  30 = 'OFF'
  29 = 'ON'
  41 = 'On'
  14 = 'OPEN'
  60 = 'ORANGE means state is active'
  10 = 'POWER OFF'
  59 = 'RED means state is active'
  3 = 'RESET'
  2 = 'REST'
  941 = 'RPC Call Status'
  47 = 'Set power intensity [%] (0..100)'
  75 = 'Stable Signal Period'
  76 = 'Stable Signal Period [ms]'
  11 = 'STATE'
  24 = 'State'
  0 = 'State: %s'
  18 = 'STATUS'
  20 = 'Status'
  21 = 'Status Description'
  5 = 'STOP'
  12 = 'SUBSTATE'
  25 = 'Substate'
  1 = 'Substate: %s'
  42 = 'Switch'
  33 = 'Time OFF = %d'
  34 = 'Time OFF Total = %d'
  83 = 'Time ON'
  86 = 'Time ON  [sec]'
  31 = 'Time ON = %d'
  32 = 'Time ON Total = %d'
  846 = 'Time since actuator was switched OFF [sec].'
  82 = 'Time since power was switched OFF [sec].'
  81 = 'Time since last ON command [sec].'
  79 = 'Time since last ON command.'
  763 = 'Total continuous time that actuator has been ON [sec].'
  80 = 'Total continuous time that power has been ON [sec].'
  85 = 'Total OFF'
  88 = 'Total OFF [sec]'
  84 = 'Total ON'
  87 = 'Total ON  [sec]'
  68 = 'Ver. %.2f'
  385 = 'Ver: %s'
  57 = 'Warmup'
  48 = 'Warmup time [sec]  (>=0). \nZero means no warmup.\n'
  49 = 'Warmup [sec]'
  410 = 'When switching actuator ON, feedback signal should become active within this period.\n'
  72 = 'When switching power ON, feedback signal should become active within this period.\n'
END_TEXTLIST

// ---- VISUs/GUI_Actuator001.TcVIS
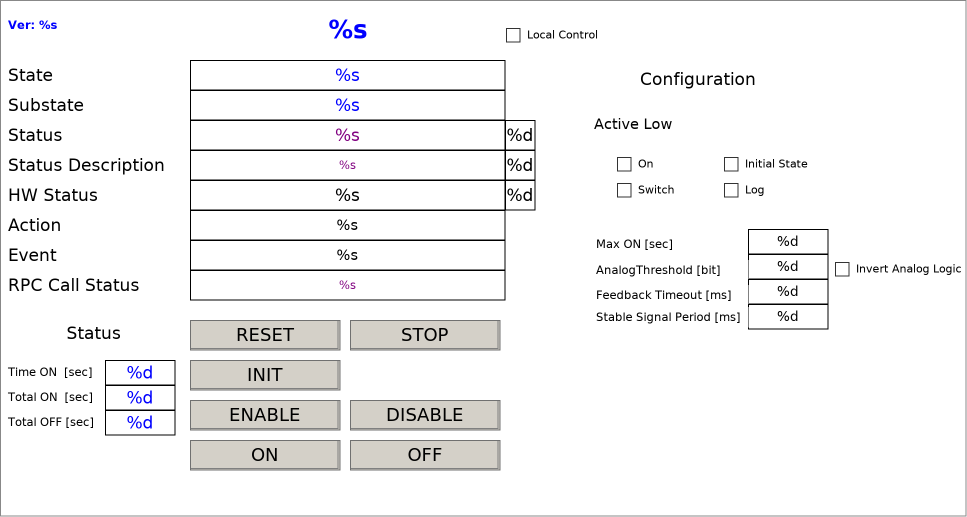
VISUALIZATION GUI_Actuator001  // 967x517
    Frame (0,0 967x517)
        shows GUI_TEMPLATE_ACTUATOR(m_Instance := MAIN.Actuator001)
END_VISUALIZATION

// ---- VISUs/GUI_Actuator002.TcVIS
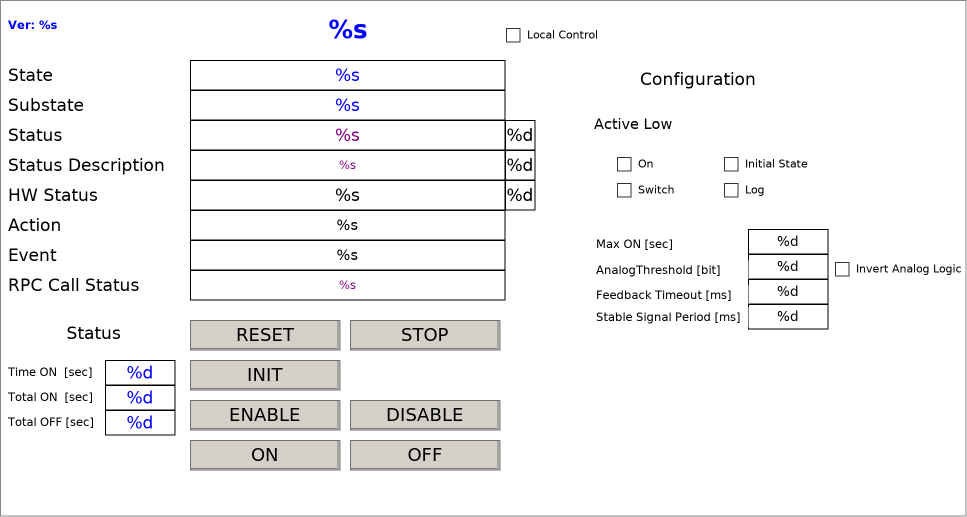
VISUALIZATION GUI_Actuator002  // 967x517
    Frame (0,0 967x517)
        shows GUI_TEMPLATE_ACTUATOR(m_Instance := MAIN.Actuator002)
END_VISUALIZATION

// ---- VISUs/GUI_Actuator003.TcVIS
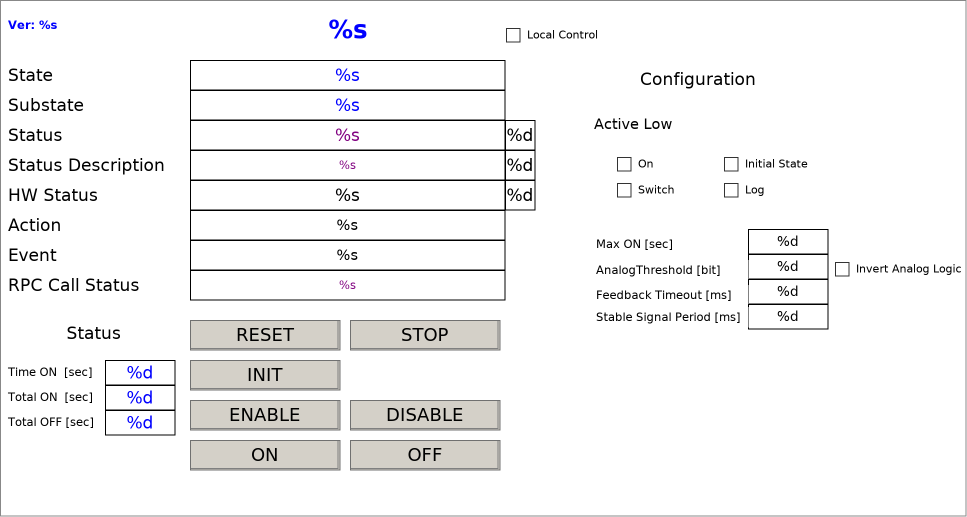
VISUALIZATION GUI_Actuator003  // 967x517
    Frame (0,0 967x517)
        shows GUI_TEMPLATE_ACTUATOR(m_Instance := MAIN.Actuator003)
END_VISUALIZATION

// ---- VISUs/GUI_Actuator004.TcVIS
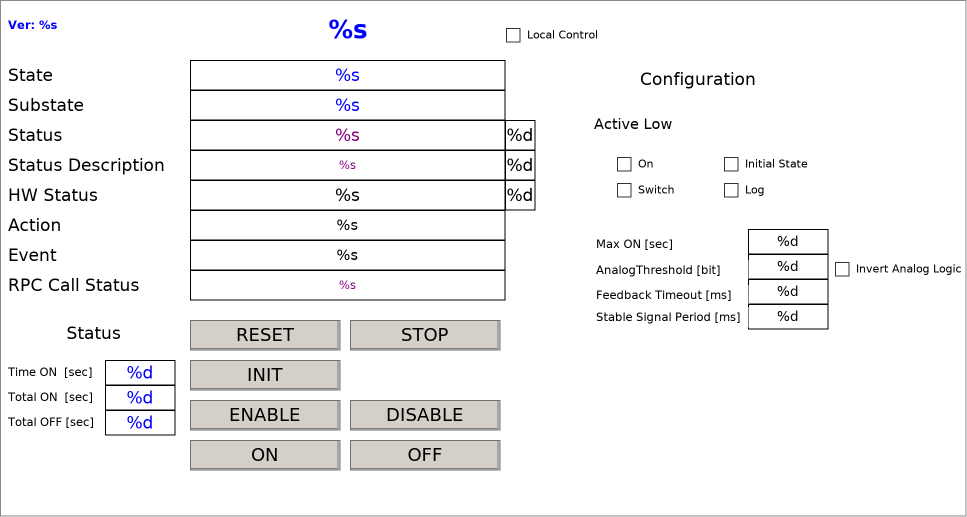
VISUALIZATION GUI_Actuator004  // 967x517
    Frame (0,0 967x517)
        shows GUI_TEMPLATE_ACTUATOR(m_Instance := MAIN.Actuator004)
END_VISUALIZATION

// ---- VISUs/Templates/GUI_TEMPLATE_ACTUATOR.TcVIS
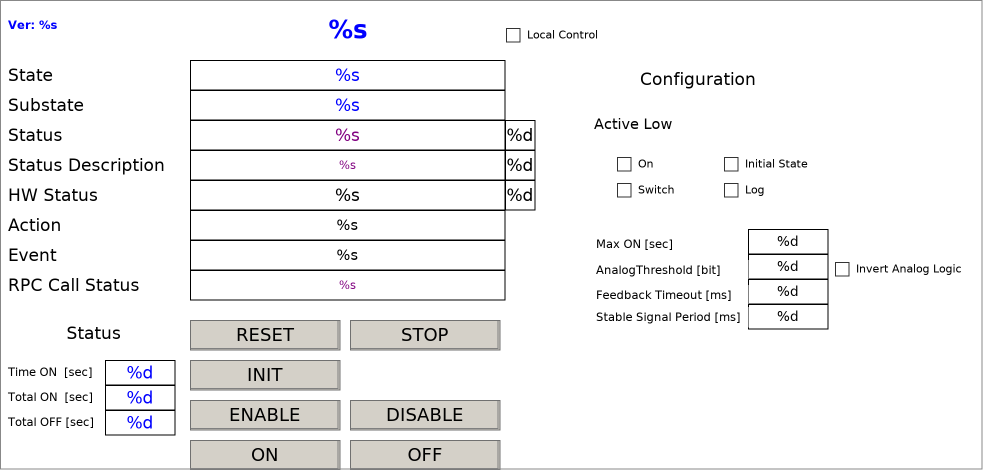
VISUALIZATION GUI_TEMPLATE_ACTUATOR  // 983x470
VAR_IN_OUT
	m_Instance:	FB_ACTUATOR;
END_VAR
    Rectangle (190,60 315x30), "%s", text variable: m_Instance.stat.sState
    Rectangle (190,90 315x30), "%s", text variable: m_Instance.stat.sSubstate
    Button (190,320 150x30), "RESET", input disabled if: (m_Instance.stat.bLocal = FALSE) <> 0
        OnMouseDown: execute { m_Instance.ctrl.nCommand := E_ACTUATOR_COMMAND.RESET; m_Instance.ctrl.bExecute := TRUE; }
    Button (190,360 150x30), "INIT", input disabled if: (m_Instance.stat.bLocal = FALSE) <> 0
        OnMouseDown: execute { m_Instance.ctrl.nCommand := E_ACTUATOR_COMMAND.INIT; m_Instance.ctrl.bExecute := TRUE; }
    Button (350,320 150x30), "STOP", input disabled if: (m_Instance.stat.bLocal = FALSE) <> 0
        OnMouseDown: execute { m_Instance.ctrl.nCommand := E_ACTUATOR_COMMAND.STOP; m_Instance.ctrl.bExecute := TRUE; }
    Button (190,400 150x30), "ENABLE", input disabled if: (m_Instance.stat.bLocal = FALSE) <> 0
        OnMouseDown: execute { m_Instance.ctrl.nCommand := E_ACTUATOR_COMMAND.ENABLE; m_Instance.ctrl.bExecute := TRUE; }
    Button (350,400 150x30), "DISABLE", input disabled if: (m_Instance.stat.bLocal = FALSE) <> 0
        OnMouseDown: execute { m_Instance.ctrl.nCommand := E_ACTUATOR_COMMAND.DISABLE; m_Instance.ctrl.bExecute := TRUE; }
    Button (190,440 150x30), "ON", input disabled if: (m_Instance.stat.bLocal = FALSE) <> 0
        OnMouseDown: execute { m_Instance.ctrl.nCommand := E_ACTUATOR_COMMAND.ON; m_Instance.ctrl.bExecute := TRUE; }
    Button (350,440 150x30), "OFF", input disabled if: (m_Instance.stat.bLocal = FALSE) <> 0
        OnMouseDown: execute { m_Instance.ctrl.nCommand := E_ACTUATOR_COMMAND.OFF; m_Instance.ctrl.bExecute := TRUE; }
    Rectangle (5,60 180x30), "State"
    Rectangle (5,90 180x30), "Substate"
    Rectangle (190,120 315x30), "%s", text variable: m_Instance.stat.sStatus
    Rectangle (190,150 315x30), "%s", text variable: m_Instance.stat.sErrorText
    Rectangle (5,120 180x30), "Status"
    Rectangle (5,150 180x30), "Status Description"
    Rectangle (190,210 315x30), "%s", text variable: m_Instance.stat.sActionDesc
    Rectangle (190,240 315x30), "%s", text variable: m_Instance.stat.sEventDesc
    Rectangle (190,180 315x30), "%s", text variable: m_Instance.stat.sHwStatus
    Rectangle (5,180 180x30), "HW Status"
    Rectangle (505,180 30x30), "%d", text variable: m_Instance.stat.nHwStatus
    Rectangle (5,210 180x30), "Action"
    Rectangle (5,240 180x30), "Event"
    Rectangle (232,12 232x35), "%s", text variable: m_Instance.cfg.sName
    Rectangle (637,64 180x30), "Configuration"
    Rectangle (591,109 126x30), "Active Low"
    Checkbox (615,149 72x30), "On", variable: m_Instance.cfg.bActiveLowOn, input disabled if: (m_Instance.stat.bLocal = FALSE) <> 0
    Checkbox (615,175 72x30), "Switch", variable: m_Instance.cfg.bActiveLowSwitch, input disabled if: (m_Instance.stat.bLocal = FALSE) <> 0
    Checkbox (833,254 150x30), "Invert Analog Logic", tooltip "If the logic is inverted, the actuator is considered to be ON, if the reading is below the threshold.", variable: m_Instance.cfg.bInvertAnalog, input disabled if: (m_Instance.stat.bLocal = FALSE) <> 0
    Rectangle (593,234 155x20), "Max ON [sec]"
    Rectangle (748,229 80x25), "%d", tooltip "Maximum allowed time for actuator to be ON [sec] (>=0). Zero means no limit.", text variable: m_Instance.cfg.nMaxOn, input disabled if: (m_Instance.stat.bLocal = FALSE) <> 0
        OnMouseDown: write the text variable via Default, min 0
    Rectangle (748,254 80x25), "%d", tooltip "Analog feedback signal threshold [bit]. If used, the threshold should be > 0.", text variable: m_Instance.cfg.nAnalogThreshold, input disabled if: (m_Instance.stat.bLocal = FALSE) <> 0
        OnMouseDown: write the text variable via Default, min 0
    Rectangle (593,260 155x20), "AnalogThreshold [bit]"
    Rectangle (748,279 80x25), "%d", tooltip "When switching actuator ON, feedback signal should become active within this period.", text variable: m_Instance.cfg.nTimeout, input disabled if: (m_Instance.stat.bLocal = FALSE) <> 0
        OnMouseDown: write the text variable via Default, min 0
    Rectangle (593,285 155x20), "Feedback Timeout [ms]"
    Checkbox (504,20 116x30), "Local Control", variable: m_Instance.stat.bLocal
    Rectangle (748,304 80x25), "%d", tooltip "A period of time [ms] that the feedback signal has to have constant value before taking its status. Minimum 10 ms.", text variable: m_Instance.cfg.nSigStablePeriod, input disabled if: (m_Instance.stat.bLocal = FALSE) <> 0
        OnMouseDown: write the text variable via Default, min 10
    Rectangle (593,307 155x20), "Stable Signal Period [ms]"
    Rectangle (48,318 92x30), "Status"
    Rectangle (105,360 70x25), "%d", tooltip "Time since last ON command [sec].", text variable: m_Instance.stat.nTimeOn
    Rectangle (105,385 70x25), "%d", tooltip "Total continuous time that actuator has been ON [sec].", text variable: m_Instance.stat.nTimeOnTotal
    Rectangle (105,410 70x25), "%d", tooltip "Time since actuator was switched OFF [sec].", text variable: m_Instance.stat.nTimeOff
    Rectangle (5,357 95x30), "Time ON [sec]"
    Rectangle (5,382 95x30), "Total ON [sec]"
    Rectangle (5,407 95x30), "Total OFF [sec]"
    Rectangle (505,120 30x30), "%d", text variable: m_Instance.stat.nStatus
    Rectangle (190,270 315x30), "%s", text variable: m_Instance.stat.sRPCErrorText
    Rectangle (5,270 180x30), "RPC Call Status"
    Rectangle (5,10 99x30), "Ver: %s", tooltip "'Actuator.library version'", text variable: stLibVersion_ESO_LDC_Actuator_Library.sVersion, input disabled if: true
    Checkbox (722,175 72x30), "Log", tooltip "If checked, logging is active.", variable: m_Instance.cfg.bLog, input disabled if: (m_Instance.stat.bLocal = FALSE) <> 0
    Checkbox (722,149 107x30), "Initial State", tooltip "If checked, switch is automatically turned ON on PLC reboot or after RESET.", variable: m_Instance.cfg.bInitialState, input disabled if: (m_Instance.stat.bLocal = FALSE) <> 0
    Rectangle (505,150 30x30), "%d", tooltip "Error code. Zero means no error.", text variable: m_Instance.stat.nErrorCode
END_VISUALIZATION
